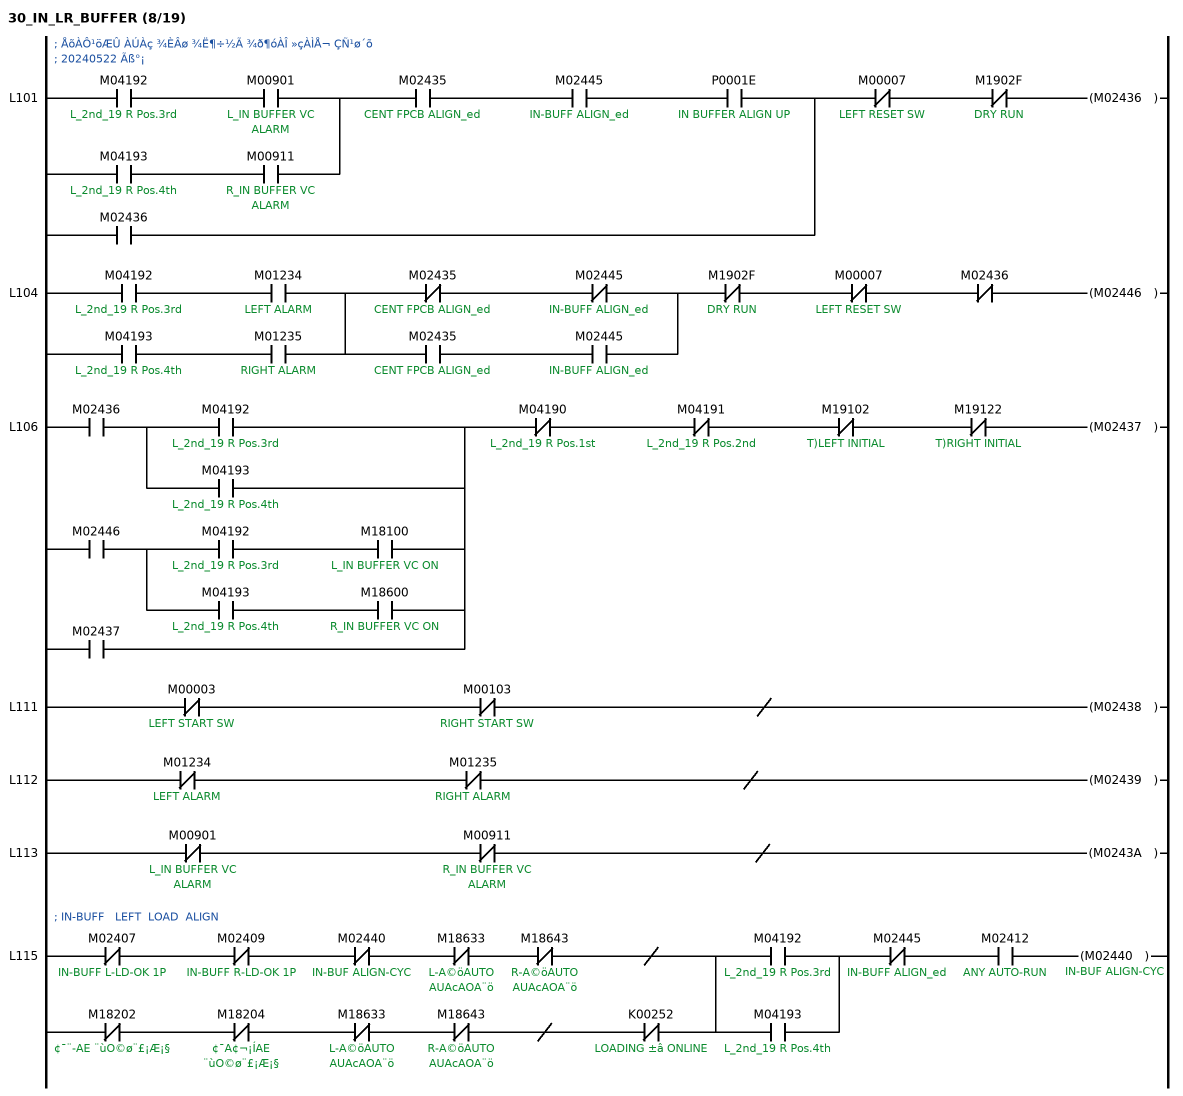
[picture p216: 30_IN_LR_BUFFER rungs L101-L115]
// ÅõÀÔ¹öÆÛ ÀÚÀç ¾ÈÂø ¾Ë¶÷½Ã ¾ð¶óÀÎ »çÀÌÅ¬ ÇÑ¹ø´õ
; L101
LOAD      M04192	// L_2nd_19 R Pos.3rd
AND       M00901	// L_IN BUFFER VC ALARM
LOAD      M04193	// L_2nd_19 R Pos.4th 
AND       M00911	// R_IN BUFFER VC ALARM
OR LOAD
AND       M02435	// CENT FPCB ALIGN_ed
AND       M02445	// IN-BUFF ALIGN_ed
AND       P0001E	// IN BUFFER ALIGN UP
OR        M02436
AND NOT   M00007	// LEFT RESET SW
AND NOT   M1902F	// DRY RUN
OUT       M02436
// output comment: 20240522 Ãß°¡
; L104
LOAD      M04192	// L_2nd_19 R Pos.3rd
AND       M01234	// LEFT ALARM
LOAD      M04193	// L_2nd_19 R Pos.4th 
AND       M01235	// RIGHT ALARM
OR LOAD
LOAD NOT  M02435	// CENT FPCB ALIGN_ed
AND NOT   M02445	// IN-BUFF ALIGN_ed
LOAD      M02435	// CENT FPCB ALIGN_ed
AND       M02445	// IN-BUFF ALIGN_ed
OR LOAD
AND LOAD
AND NOT   M1902F	// DRY RUN
AND NOT   M00007	// LEFT RESET SW
AND NOT   M02436
OUT       M02446
; L106
LOAD      M02436
LOAD      M04192	// L_2nd_19 R Pos.3rd
OR        M04193	// L_2nd_19 R Pos.4th 
AND LOAD
LOAD      M02446
LOAD      M04192	// L_2nd_19 R Pos.3rd
AND       M18100	// L_IN BUFFER VC ON
LOAD      M04193	// L_2nd_19 R Pos.4th 
AND       M18600	// R_IN BUFFER VC ON
OR LOAD
AND LOAD
OR LOAD
OR        M02437
AND NOT   M04190	// L_2nd_19 R Pos.1st 
AND NOT   M04191	// L_2nd_19 R Pos.2nd
AND NOT   M19102	// T)LEFT INITIAL
AND NOT   M19122	// T)RIGHT INITIAL
OUT       M02437
; L111
LOAD NOT  M00003	// LEFT START SW
AND NOT   M00103	// RIGHT START SW
NOT
OUT       M02438
; L112
LOAD NOT  M01234	// LEFT ALARM
AND NOT   M01235	// RIGHT ALARM
NOT
OUT       M02439
; L113
LOAD NOT  M00901	// L_IN BUFFER VC ALARM
AND NOT   M00911	// R_IN BUFFER VC ALARM
NOT
OUT       M0243A
// IN-BUFF   LEFT  LOAD  ALIGN
; L115
LOAD NOT  M02407	// IN-BUFF L-LD-OK 1P
AND NOT   M02409	// IN-BUFF R-LD-OK 1P
AND NOT   M02440	// IN-BUF ALIGN-CYC
AND NOT   M18633	// L-A©öAUTO AUAcAOA¨ö
AND NOT   M18643	// R-A©öAUTO AUAcAOA¨ö
NOT
LOAD NOT  M18202	// ¢¯¨­AE ¨ùO©ø¨£¡Æ¡§
AND NOT   M18204	// ¢¯A¢¬¡ÍAE ¨ùO©ø¨£¡Æ¡§
AND NOT   M18633	// L-A©öAUTO AUAcAOA¨ö
AND NOT   M18643	// R-A©öAUTO AUAcAOA¨ö
NOT
AND NOT   K00252	// LOADING ±â ONLINE
OR LOAD
LOAD      M04192	// L_2nd_19 R Pos.3rd
OR        M04193	// L_2nd_19 R Pos.4th 
AND LOAD
AND NOT   M02445	// IN-BUFF ALIGN_ed
AND       M02412	// ANY AUTO-RUN
OUT       M02440	// IN-BUF ALIGN-CYC

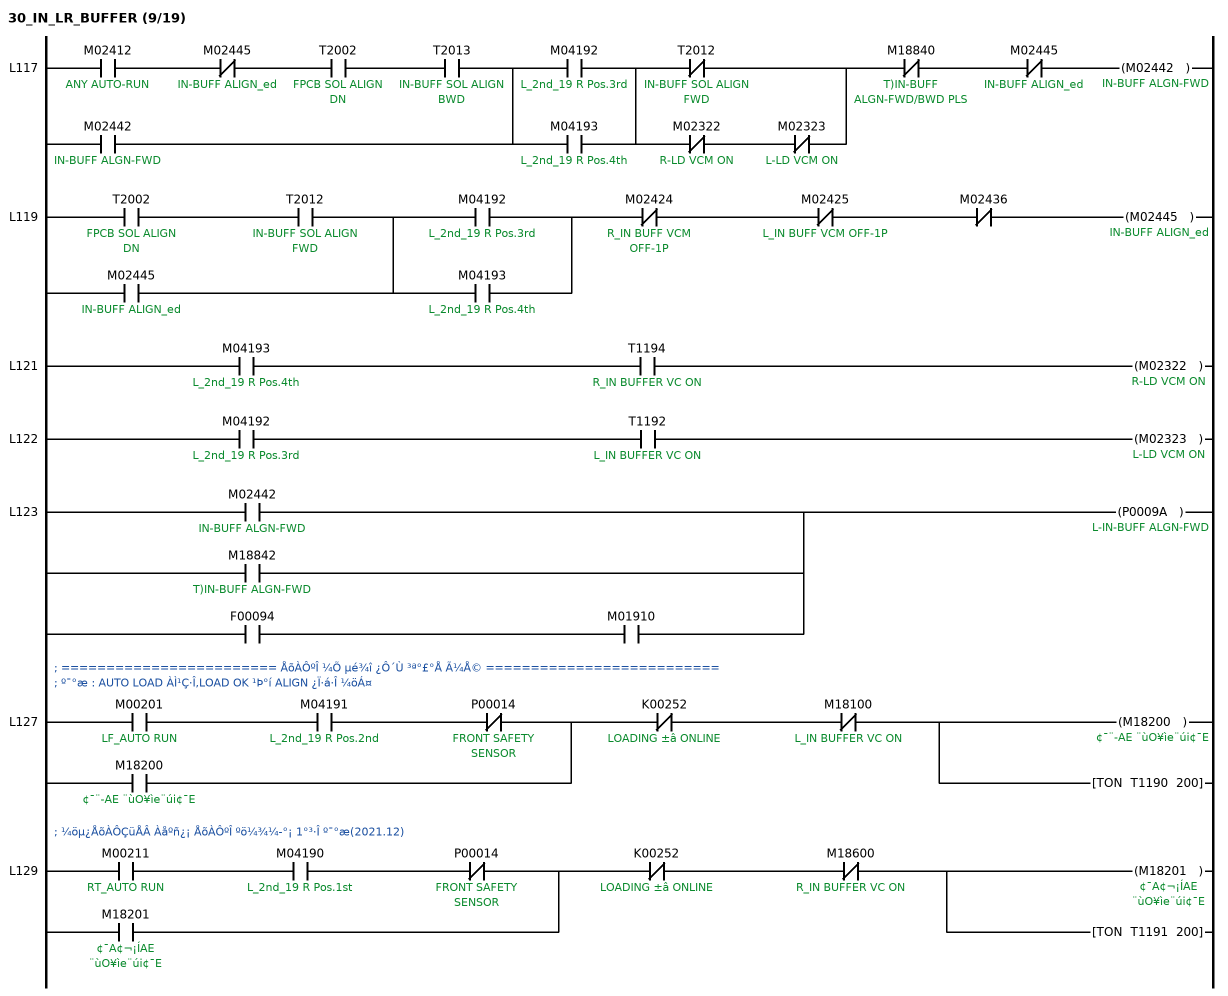
; L117
LOAD      M02412	// ANY AUTO-RUN
AND NOT   M02445	// IN-BUFF ALIGN_ed
AND       T2002	// FPCB SOL ALIGN        DN
AND       T2013	// IN-BUFF SOL ALIGN BWD
OR        M02442	// IN-BUFF ALGN-FWD
LOAD      M04192	// L_2nd_19 R Pos.3rd
OR        M04193	// L_2nd_19 R Pos.4th 
AND LOAD
LOAD NOT  T2012	// IN-BUFF SOL ALIGN FWD
LOAD NOT  M02322	// R-LD VCM ON
AND NOT   M02323	// L-LD VCM ON
OR LOAD
AND LOAD
AND NOT   M18840	// T)IN-BUFF ALGN-FWD/BWD PLS
AND NOT   M02445	// IN-BUFF ALIGN_ed
OUT       M02442	// IN-BUFF ALGN-FWD
; L119
LOAD      T2002	// FPCB SOL ALIGN        DN
AND       T2012	// IN-BUFF SOL ALIGN FWD
OR        M02445	// IN-BUFF ALIGN_ed
LOAD      M04192	// L_2nd_19 R Pos.3rd
OR        M04193	// L_2nd_19 R Pos.4th 
AND LOAD
AND NOT   M02424	// R_IN BUFF VCM OFF-1P
AND NOT   M02425	// L_IN BUFF VCM OFF-1P
AND NOT   M02436
OUT       M02445	// IN-BUFF ALIGN_ed
; L121
LOAD      M04193	// L_2nd_19 R Pos.4th 
AND       T1194	// R_IN BUFFER VC ON
OUT       M02322	// R-LD VCM ON
; L122
LOAD      M04192	// L_2nd_19 R Pos.3rd
AND       T1192	// L_IN BUFFER VC ON
OUT       M02323	// L-LD VCM ON
; L123
LOAD      M02442	// IN-BUFF ALGN-FWD
OR        M18842	// T)IN-BUFF ALGN-FWD
LOAD      F00094
AND       M01910
OR LOAD
OUT       P0009A	// L-IN-BUFF ALGN-FWD
// ======================== ÅõÀÔºÎ ¼Õ µé¾î ¿Ô´Ù ³ª°£°Å Ã¼Å© ==========================
// 
// º¯°æ : AUTO LOAD ÀÌ¹Ç·Î,LOAD OK ¹Þ°í ALIGN ¿Ï·á·Î ¼öÁ¤
; L127
LOAD      M00201	// LF_AUTO RUN
AND       M04191	// L_2nd_19 R Pos.2nd
AND NOT   P00014	// FRONT SAFETY SENSOR
OR        M18200	// ¢¯¨­AE ¨ùO¥ìe¨úi¢¯E
AND NOT   K00252	// LOADING ±â ONLINE
AND NOT   M18100	// L_IN BUFFER VC ON
OUT       M18200	// ¢¯¨­AE ¨ùO¥ìe¨úi¢¯E
TON       T1190 200
; L129
LOAD      M00211	// RT_AUTO RUN
AND       M04190	// L_2nd_19 R Pos.1st 
AND NOT   P00014	// FRONT SAFETY SENSOR
OR        M18201	// ¢¯A¢¬¡ÍAE ¨ùO¥ìe¨úi¢¯E
AND NOT   K00252	// LOADING ±â ONLINE
AND NOT   M18600	// R_IN BUFFER VC ON
OUT       M18201	// ¢¯A¢¬¡ÍAE ¨ùO¥ìe¨úi¢¯E
TON       T1191 200
// output comment: ¼öµ¿ÅõÀÔÇüÅÂ Àåºñ¿¡ ÅõÀÔºÎ ºö¼¾¼­°¡ 1°³·Î º¯°æ(2021.12)

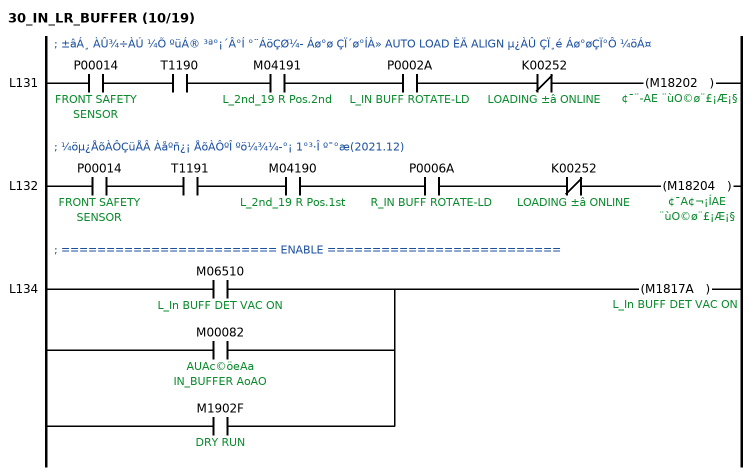
; L131
LOAD      P00014	// FRONT SAFETY SENSOR
AND       T1190
AND       M04191	// L_2nd_19 R Pos.2nd
AND       P0002A	// L_IN BUFF ROTATE-LD
AND NOT   K00252	// LOADING ±â ONLINE
OUT       M18202	// ¢¯¨­AE ¨ùO©ø¨£¡Æ¡§
// output comment: ±âÁ¸ ÀÛ¾÷ÀÚ ¼Õ ºüÁ® ³ª°¡´Â°Í °¨ÁöÇØ¼­ Áø°ø ÇÏ´ø°ÍÀ» AUTO LOAD ÈÄ ALIGN µ¿ÀÛ ÇÏ¸é Áø°øÇÏ°Ô ¼öÁ¤
; L132
LOAD      P00014	// FRONT SAFETY SENSOR
AND       T1191
AND       M04190	// L_2nd_19 R Pos.1st 
AND       P0006A	// R_IN BUFF ROTATE-LD
AND NOT   K00252	// LOADING ±â ONLINE
OUT       M18204	// ¢¯A¢¬¡ÍAE ¨ùO©ø¨£¡Æ¡§
// output comment: ¼öµ¿ÅõÀÔÇüÅÂ Àåºñ¿¡ ÅõÀÔºÎ ºö¼¾¼­°¡ 1°³·Î º¯°æ(2021.12)
// ======================== ENABLE ==========================
; L134
LOAD      M06510	// L_In BUFF DET VAC ON
OR        M00082	// AUAc©öeAa IN_BUFFER AoAO 
OR        M1902F	// DRY RUN
OUT       M1817A	// L_In BUFF DET VAC ON

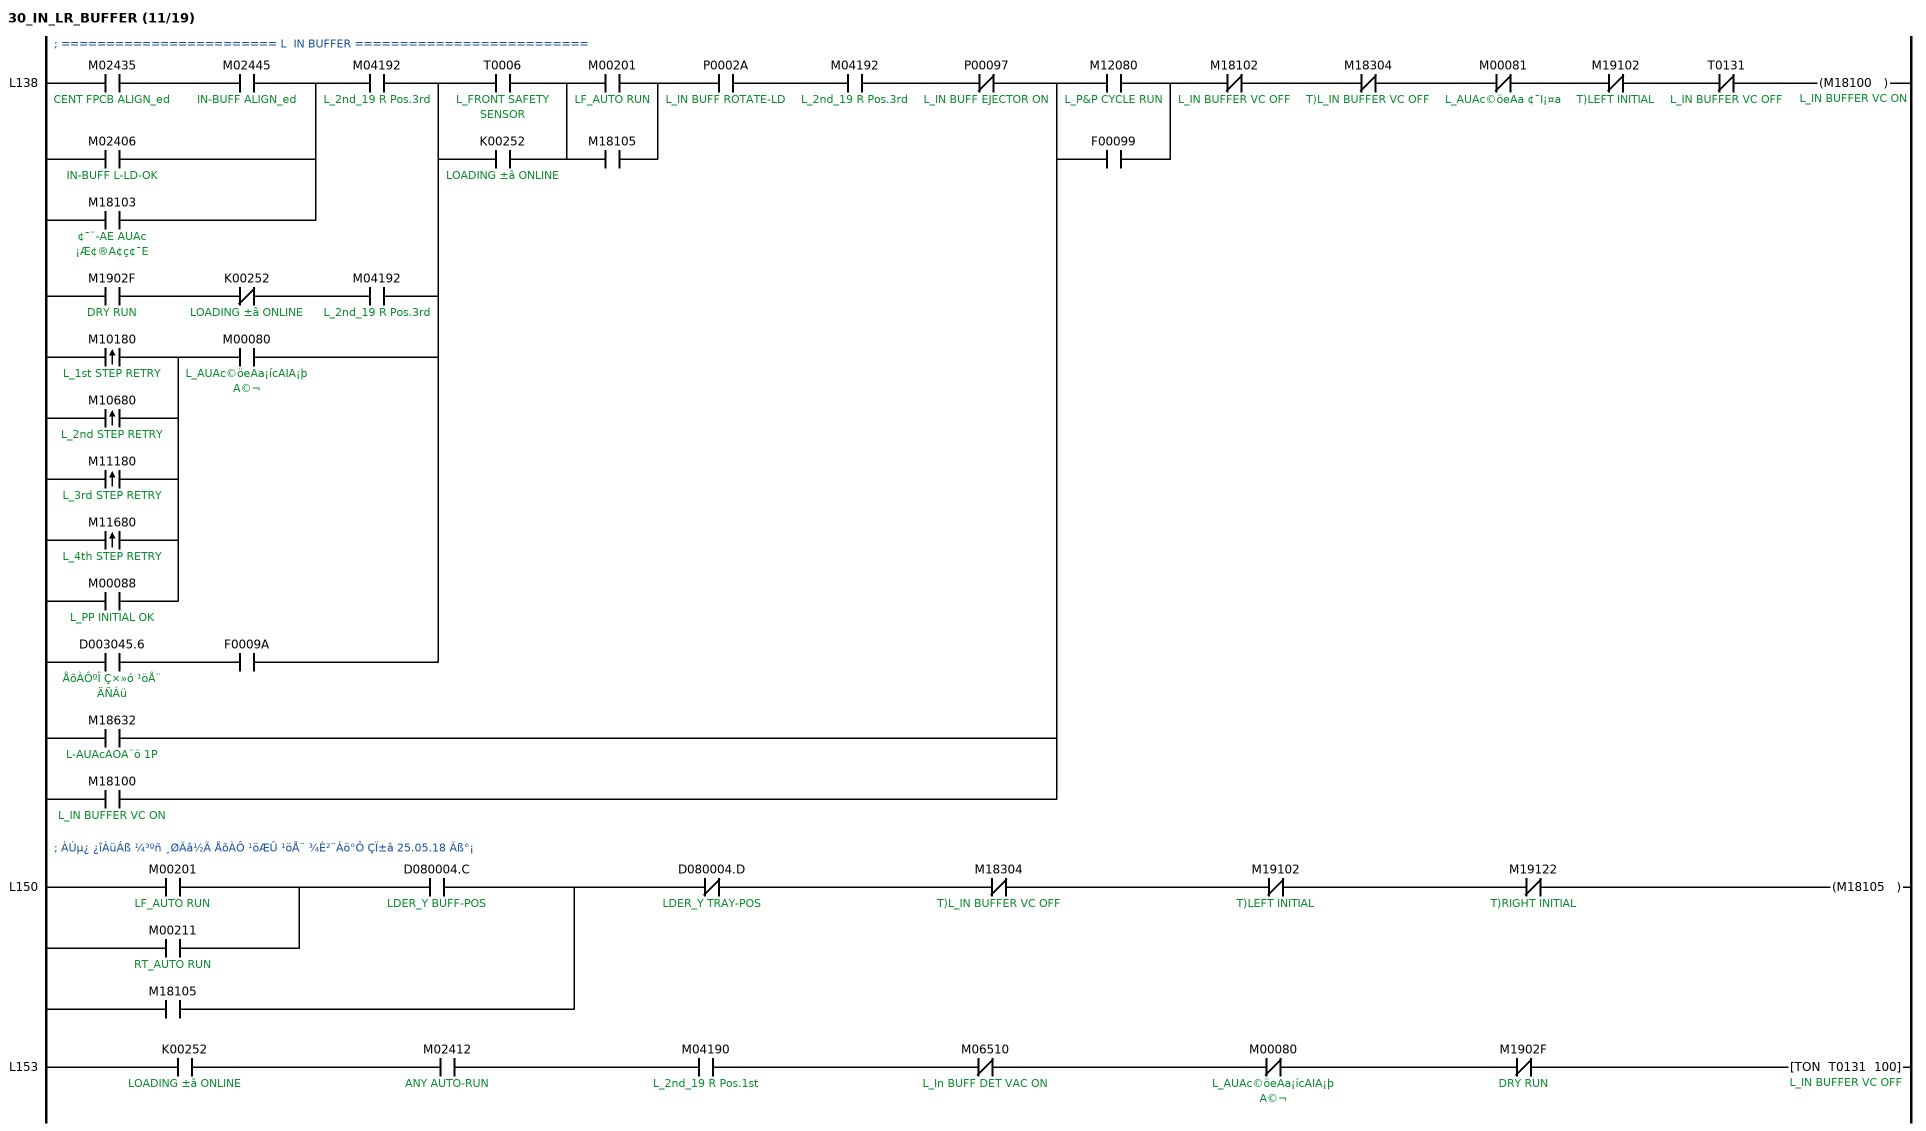
// ======================== L  IN BUFFER ==========================
; L138
LOAD      M02435	// CENT FPCB ALIGN_ed
AND       M02445	// IN-BUFF ALIGN_ed
OR        M02406	// IN-BUFF L-LD-OK
OR        M18103	// ¢¯¨­AE AUAc ¡Æ¢®A¢ç¢¯E
AND       M04192	// L_2nd_19 R Pos.3rd
LOAD      M1902F	// DRY RUN
AND NOT   K00252	// LOADING ±â ONLINE
AND       M04192	// L_2nd_19 R Pos.3rd
OR LOAD
LOADP     M10180	// L_1st STEP RETRY
ORP       M10680	// L_2nd STEP RETRY
ORP       M11180	// L_3rd STEP RETRY
ORP       M11680	// L_4th STEP RETRY
OR        M00088	// L_PP INITIAL OK
AND       M00080	// L_AUAc©öeAa¡ícAIA¡þA©¬
OR LOAD
LOAD      D003045.6	// ÅõÀÔºÎ Ç×»ó ¹öÅ¨ ÄÑÁü
AND       F0009A
OR LOAD
LOAD      T0006	// L_FRONT SAFETY SENSOR
OR        K00252	// LOADING ±â ONLINE
AND LOAD
LOAD      M00201	// LF_AUTO RUN
OR        M18105
AND LOAD
AND       P0002A	// L_IN BUFF ROTATE-LD
AND       M04192	// L_2nd_19 R Pos.3rd
AND NOT   P00097	// L_IN BUFF EJECTOR ON
OR        M18632	// L-AUAcAOA¨ö 1P
OR        M18100	// L_IN BUFFER VC ON
LOAD      M12080	// L_P&P CYCLE RUN
OR        F00099
AND LOAD
AND NOT   M18102	// L_IN BUFFER VC OFF
AND NOT   M18304	// T)L_IN BUFFER VC OFF
AND NOT   M00081	// L_AUAc©öeAa ¢¯I¡¤a
AND NOT   M19102	// T)LEFT INITIAL
AND NOT   T0131	// L_IN BUFFER VC OFF
OUT       M18100	// L_IN BUFFER VC ON
; L150
LOAD      M00201	// LF_AUTO RUN
OR        M00211	// RT_AUTO RUN
AND       D080004.C	// LDER_Y BUFF-POS
OR        M18105
AND NOT   D080004.D	// LDER_Y TRAY-POS
AND NOT   M18304	// T)L_IN BUFFER VC OFF
AND NOT   M19102	// T)LEFT INITIAL
AND NOT   M19122	// T)RIGHT INITIAL
OUT       M18105
// output comment: ÀÚµ¿ ¿îÀüÁß ¼³ºñ ¸ØÃâ½Ã ÅõÀÔ ¹öÆÛ ¹öÅ¨ ¾È²¨Áö°Ô ÇÏ±â 25.05.18 Ãß°¡
; L153
LOAD      K00252	// LOADING ±â ONLINE
AND       M02412	// ANY AUTO-RUN
AND       M04190	// L_2nd_19 R Pos.1st 
AND NOT   M06510	// L_In BUFF DET VAC ON
AND NOT   M00080	// L_AUAc©öeAa¡ícAIA¡þA©¬
AND NOT   M1902F	// DRY RUN
TON       T0131 100	// L_IN BUFFER VC OFF

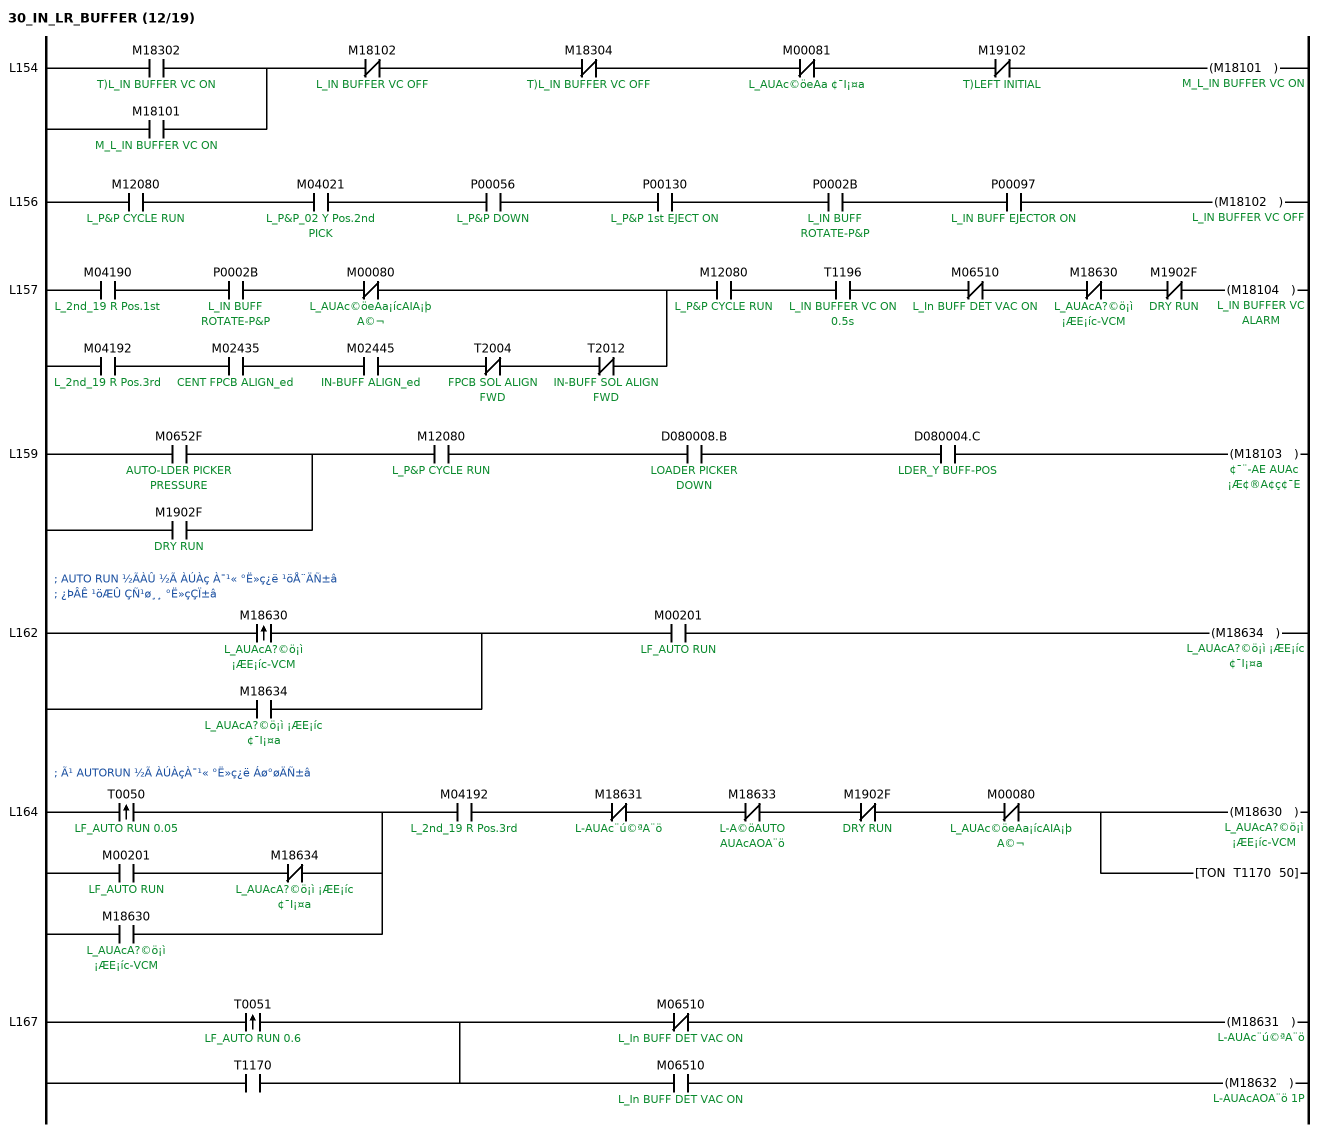
; L154
LOAD      M18302	// T)L_IN BUFFER VC ON
OR        M18101	// M_L_IN BUFFER VC ON
AND NOT   M18102	// L_IN BUFFER VC OFF
AND NOT   M18304	// T)L_IN BUFFER VC OFF
AND NOT   M00081	// L_AUAc©öeAa ¢¯I¡¤a
AND NOT   M19102	// T)LEFT INITIAL
OUT       M18101	// M_L_IN BUFFER VC ON
; L156
LOAD      M12080	// L_P&P CYCLE RUN
AND       M04021	// L_P&P_02 Y Pos.2nd PICK
AND       P00056	// L_P&P DOWN
AND       P00130	// L_P&P 1st EJECT ON
AND       P0002B	// L_IN BUFF ROTATE-P&P
AND       P00097	// L_IN BUFF EJECTOR ON
OUT       M18102	// L_IN BUFFER VC OFF
; L157
LOAD      M04190	// L_2nd_19 R Pos.1st 
AND       P0002B	// L_IN BUFF ROTATE-P&P
AND NOT   M00080	// L_AUAc©öeAa¡ícAIA¡þA©¬
LOAD      M04192	// L_2nd_19 R Pos.3rd
AND       M02435	// CENT FPCB ALIGN_ed
AND       M02445	// IN-BUFF ALIGN_ed
AND NOT   T2004	// FPCB SOL ALIGN         FWD
AND NOT   T2012	// IN-BUFF SOL ALIGN FWD
OR LOAD
AND       M12080	// L_P&P CYCLE RUN
AND       T1196	// L_IN BUFFER VC ON 0.5s
AND NOT   M06510	// L_In BUFF DET VAC ON
AND NOT   M18630	// L_AUAcA?©ö¡ì ¡ÆE¡íc-VCM
AND NOT   M1902F	// DRY RUN
OUT       M18104	// L_IN BUFFER VC ALARM
; L159
LOAD      M0652F	// AUTO-LDER PICKER PRESSURE
OR        M1902F	// DRY RUN
AND       M12080	// L_P&P CYCLE RUN
AND       D080008.B	// LOADER PICKER DOWN
AND       D080004.C	// LDER_Y BUFF-POS
OUT       M18103	// ¢¯¨­AE AUAc ¡Æ¢®A¢ç¢¯E
// AUTO RUN ½ÃÀÛ ½Ã ÀÚÀç À¯¹« °Ë»ç¿ë ¹öÅ¨ÄÑ±â
; L162
LOADP     M18630	// L_AUAcA?©ö¡ì ¡ÆE¡íc-VCM
OR        M18634	// L_AUAcA?©ö¡ì ¡ÆE¡íc ¢¯I¡¤a
AND       M00201	// LF_AUTO RUN
OUT       M18634	// L_AUAcA?©ö¡ì ¡ÆE¡íc ¢¯I¡¤a
// output comment: ¿ÞÂÊ ¹öÆÛ ÇÑ¹ø¸¸ °Ë»çÇÏ±â
; L164
LOADP     T0050	// LF_AUTO RUN 0.05
LOAD      M00201	// LF_AUTO RUN
AND NOT   M18634	// L_AUAcA?©ö¡ì ¡ÆE¡íc ¢¯I¡¤a
OR LOAD
OR        M18630	// L_AUAcA?©ö¡ì ¡ÆE¡íc-VCM
AND       M04192	// L_2nd_19 R Pos.3rd
AND NOT   M18631	// L-AUAc¨ú©ªA¨ö
AND NOT   M18633	// L-A©öAUTO AUAcAOA¨ö
AND NOT   M1902F	// DRY RUN
AND NOT   M00080	// L_AUAc©öeAa¡ícAIA¡þA©¬
OUT       M18630	// L_AUAcA?©ö¡ì ¡ÆE¡íc-VCM
TON       T1170 50
// output comment: Ã¹ AUTORUN ½Ã ÀÚÀçÀ¯¹« °Ë»ç¿ë Áø°øÄÑ±â
; L167
LOADP     T0051	// LF_AUTO RUN 0.6
OR        T1170
MPUSH
AND NOT   M06510	// L_In BUFF DET VAC ON
OUT       M18631	// L-AUAc¨ú©ªA¨ö
MPOP
AND       M06510	// L_In BUFF DET VAC ON
OUT       M18632	// L-AUAcAOA¨ö 1P

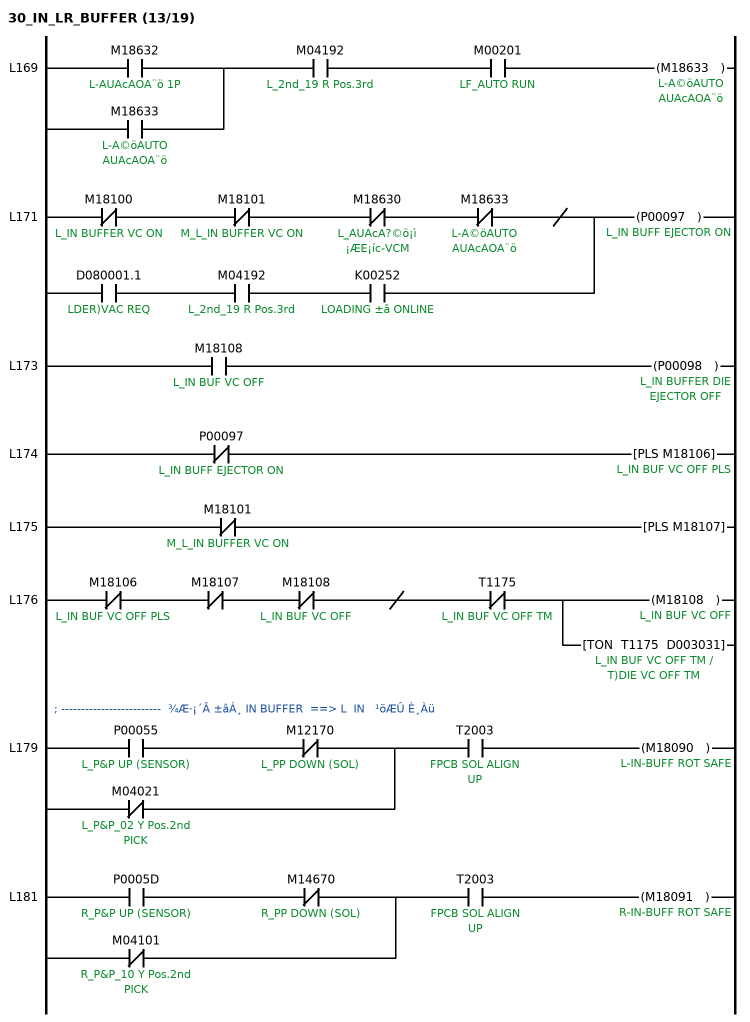
; L169
LOAD      M18632	// L-AUAcAOA¨ö 1P
OR        M18633	// L-A©öAUTO AUAcAOA¨ö
AND       M04192	// L_2nd_19 R Pos.3rd
AND       M00201	// LF_AUTO RUN
OUT       M18633	// L-A©öAUTO AUAcAOA¨ö
; L171
LOAD NOT  M18100	// L_IN BUFFER VC ON
AND NOT   M18101	// M_L_IN BUFFER VC ON
AND NOT   M18630	// L_AUAcA?©ö¡ì ¡ÆE¡íc-VCM
AND NOT   M18633	// L-A©öAUTO AUAcAOA¨ö
NOT
LOAD      D080001.1	// LDER)VAC REQ
AND       M04192	// L_2nd_19 R Pos.3rd
AND       K00252	// LOADING ±â ONLINE
OR LOAD
OUT       P00097	// L_IN BUFF EJECTOR ON
; L173
LOAD      M18108	// L_IN BUF VC OFF
OUT       P00098	// L_IN BUFFER DIE EJECTOR OFF
; L174
LOAD NOT  P00097	// L_IN BUFF EJECTOR ON
OUTP      M18106	// L_IN BUF VC OFF PLS
; L175
LOAD NOT  M18101	// M_L_IN BUFFER VC ON
OUTP      M18107
; L176
LOAD NOT  M18106	// L_IN BUF VC OFF PLS
AND NOT   M18107
AND NOT   M18108	// L_IN BUF VC OFF
NOT
AND NOT   T1175	// L_IN BUF VC OFF TM
OUT       M18108	// L_IN BUF VC OFF
TON       T1175 D003031	// L_IN BUF VC OFF TM / T)DIE VC OFF TM
// -------------------------  ¾Æ·¡´Â ±âÁ¸ IN BUFFER  ==> L  IN   ¹öÆÛ È¸Àü
; L179
LOAD      P00055	// L_P&P UP (SENSOR)
AND NOT   M12170	// L_PP DOWN (SOL)
OR NOT    M04021	// L_P&P_02 Y Pos.2nd PICK
AND       T2003	// FPCB SOL ALIGN         UP
OUT       M18090	// L-IN-BUFF ROT SAFE
; L181
LOAD      P0005D	// R_P&P UP (SENSOR)
AND NOT   M14670	// R_PP DOWN (SOL)
OR NOT    M04101	// R_P&P_10 Y Pos.2nd PICK
AND       T2003	// FPCB SOL ALIGN         UP
OUT       M18091	// R-IN-BUFF ROT SAFE

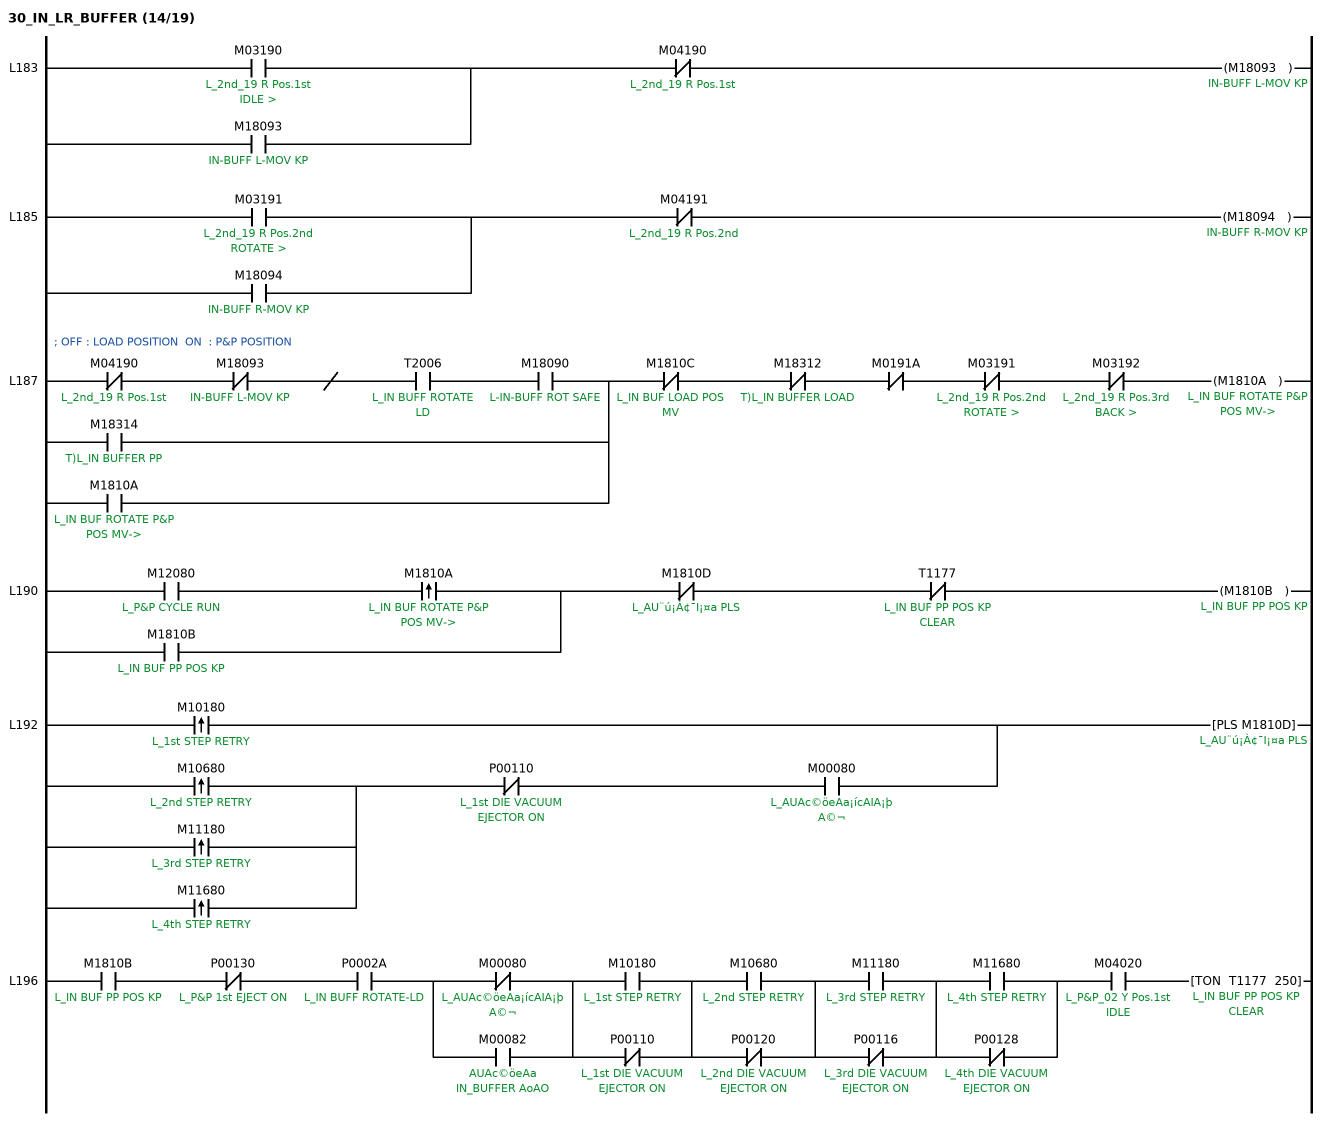
; L183
LOAD      M03190	// L_2nd_19 R Pos.1st IDLE >
OR        M18093	// IN-BUFF L-MOV KP
AND NOT   M04190	// L_2nd_19 R Pos.1st 
OUT       M18093	// IN-BUFF L-MOV KP
; L185
LOAD      M03191	// L_2nd_19 R Pos.2nd ROTATE >
OR        M18094	// IN-BUFF R-MOV KP
AND NOT   M04191	// L_2nd_19 R Pos.2nd
OUT       M18094	// IN-BUFF R-MOV KP
; L187
LOAD NOT  M04190	// L_2nd_19 R Pos.1st 
AND NOT   M18093	// IN-BUFF L-MOV KP
NOT
AND       T2006	// L_IN BUFF ROTATE     LD
AND       M18090	// L-IN-BUFF ROT SAFE
OR        M18314	// T)L_IN BUFFER PP
OR        M1810A	// L_IN BUF ROTATE P&P POS MV->
AND NOT   M1810C	// L_IN BUF LOAD POS MV
AND NOT   M18312	// T)L_IN BUFFER LOAD
AND NOT   M0191A
AND NOT   M03191	// L_2nd_19 R Pos.2nd ROTATE >
AND NOT   M03192	// L_2nd_19 R Pos.3rd BACK >
OUT       M1810A	// L_IN BUF ROTATE P&P POS MV->
// output comment: OFF : LOAD POSITION  ON  : P&P POSITION
; L190
LOAD      M12080	// L_P&P CYCLE RUN
ANDP      M1810A	// L_IN BUF ROTATE P&P POS MV->
OR        M1810B	// L_IN BUF PP POS KP
AND NOT   M1810D	// L_AU¨ú¡À¢¯I¡¤a PLS
AND NOT   T1177	// L_IN BUF PP POS KP CLEAR
OUT       M1810B	// L_IN BUF PP POS KP
; L192
LOADP     M10180	// L_1st STEP RETRY
LOADP     M10680	// L_2nd STEP RETRY
ORP       M11180	// L_3rd STEP RETRY
ORP       M11680	// L_4th STEP RETRY
AND NOT   P00110	// L_1st DIE VACUUM EJECTOR ON
AND       M00080	// L_AUAc©öeAa¡ícAIA¡þA©¬
OR LOAD
OUTP      M1810D	// L_AU¨ú¡À¢¯I¡¤a PLS
; L196
LOAD      M1810B	// L_IN BUF PP POS KP
AND NOT   P00130	// L_P&P 1st EJECT ON
AND       P0002A	// L_IN BUFF ROTATE-LD
LOAD NOT  M00080	// L_AUAc©öeAa¡ícAIA¡þA©¬
OR        M00082	// AUAc©öeAa IN_BUFFER AoAO 
AND LOAD
LOAD      M10180	// L_1st STEP RETRY
OR NOT    P00110	// L_1st DIE VACUUM EJECTOR ON
AND LOAD
LOAD      M10680	// L_2nd STEP RETRY
OR NOT    P00120	// L_2nd DIE VACUUM EJECTOR ON
AND LOAD
LOAD      M11180	// L_3rd STEP RETRY
OR NOT    P00116	// L_3rd DIE VACUUM EJECTOR ON
AND LOAD
LOAD      M11680	// L_4th STEP RETRY
OR NOT    P00128	// L_4th DIE VACUUM EJECTOR ON
AND LOAD
AND       M04020	// L_P&P_02 Y Pos.1st IDLE
TON       T1177 250	// L_IN BUF PP POS KP CLEAR

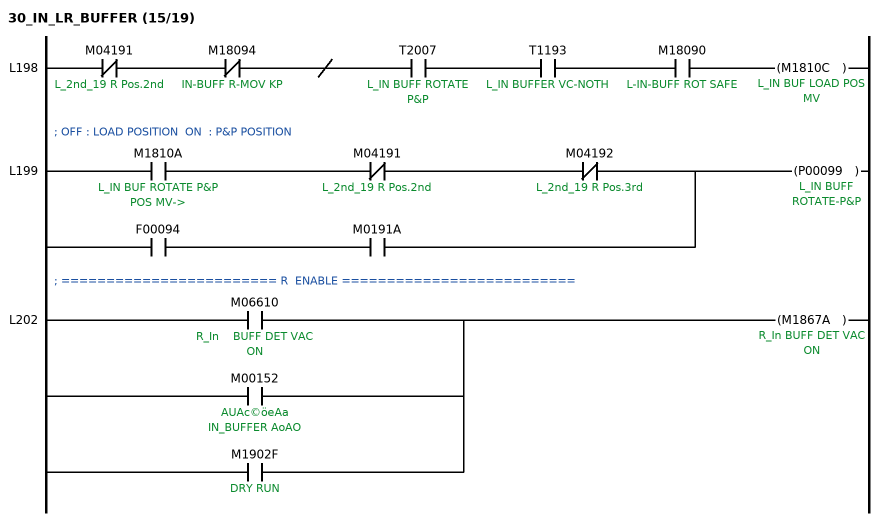
; L198
LOAD NOT  M04191	// L_2nd_19 R Pos.2nd
AND NOT   M18094	// IN-BUFF R-MOV KP
NOT
AND       T2007	// L_IN BUFF ROTATE      P&P
AND       T1193	// L_IN BUFFER VC-NOTH
AND       M18090	// L-IN-BUFF ROT SAFE
OUT       M1810C	// L_IN BUF LOAD POS MV
; L199
LOAD      M1810A	// L_IN BUF ROTATE P&P POS MV->
AND NOT   M04191	// L_2nd_19 R Pos.2nd
AND NOT   M04192	// L_2nd_19 R Pos.3rd
LOAD      F00094
AND       M0191A
OR LOAD
OUT       P00099	// L_IN BUFF ROTATE-P&P
// output comment: OFF : LOAD POSITION  ON  : P&P POSITION
// ======================== R  ENABLE ==========================
; L202
LOAD      M06610	// R_In    BUFF DET VAC ON
OR        M00152	// AUAc©öeAa IN_BUFFER AoAO 
OR        M1902F	// DRY RUN
OUT       M1867A	// R_In BUFF DET VAC ON

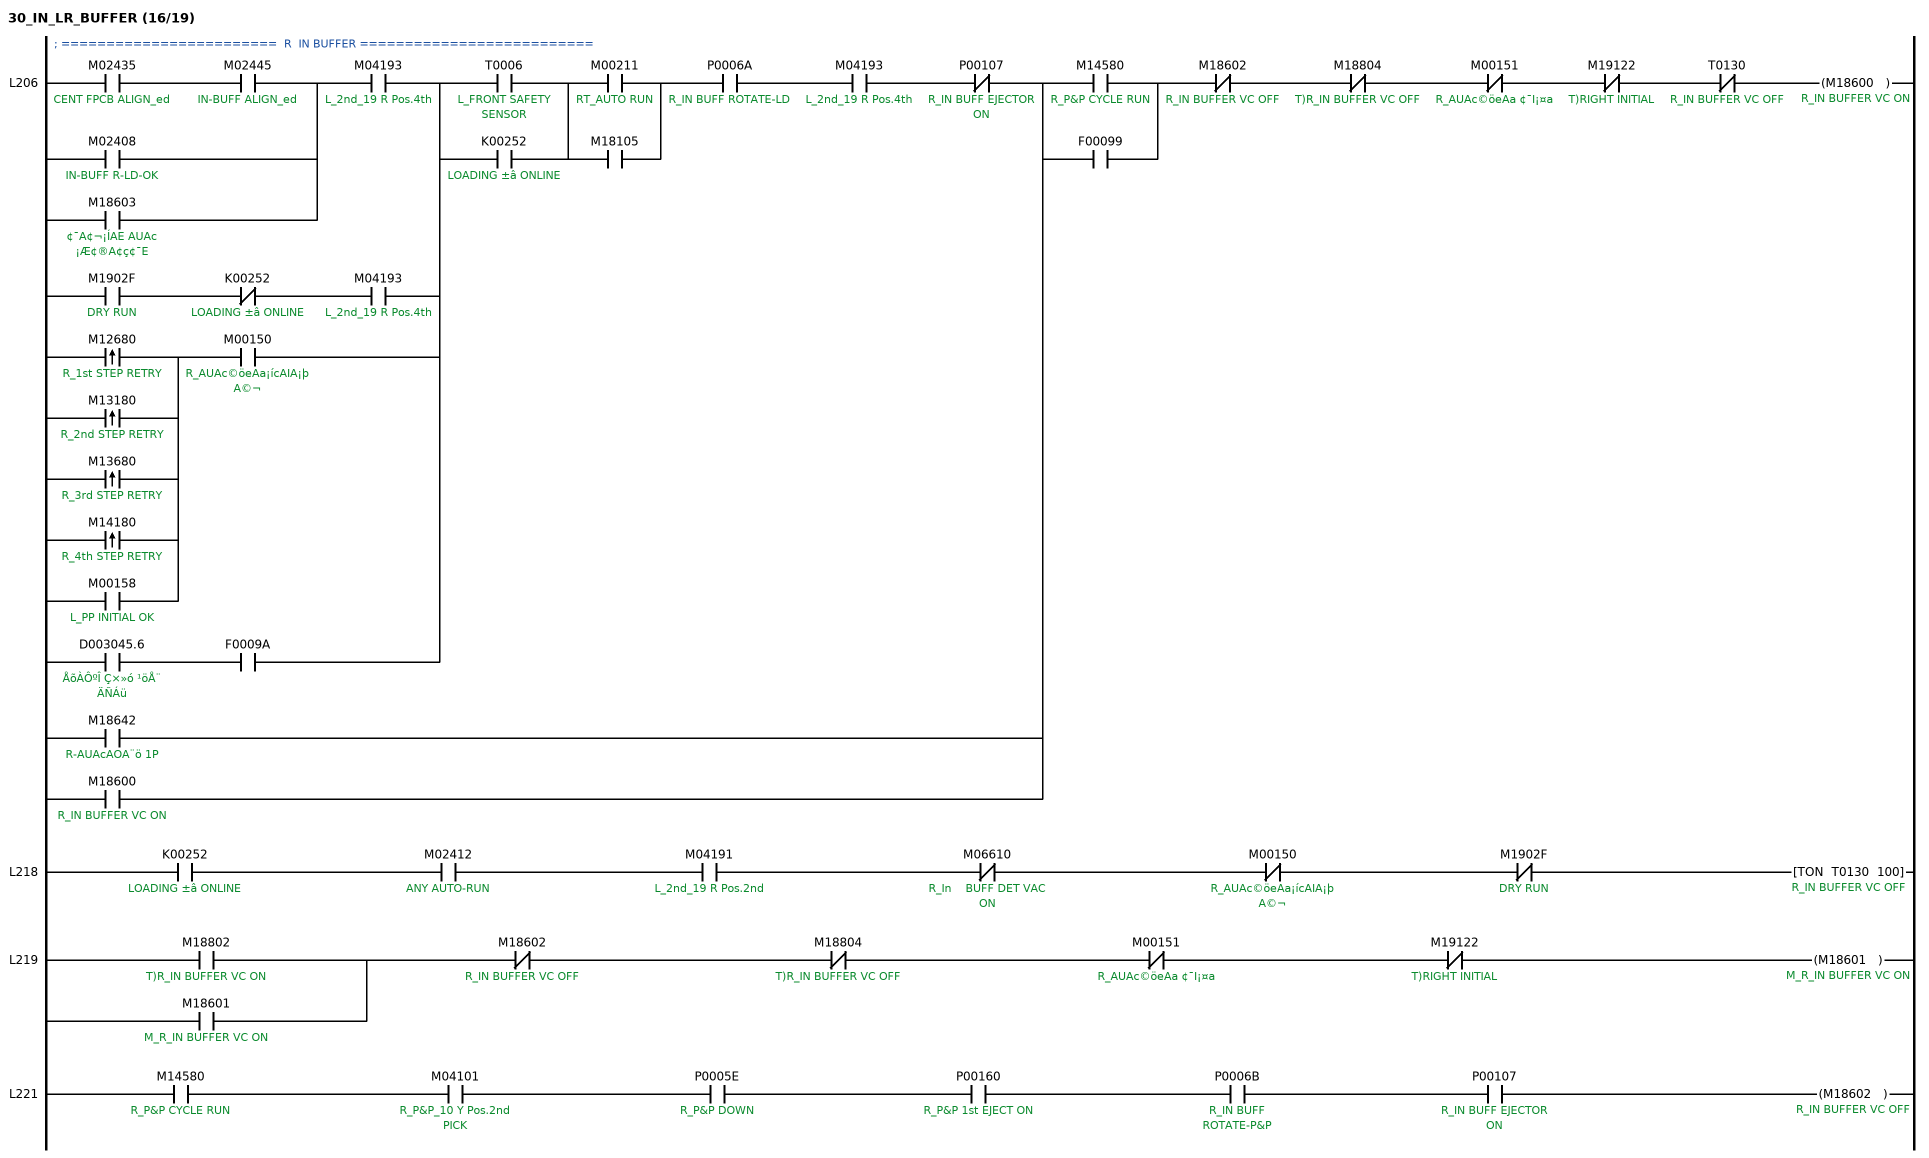
// ========================  R  IN BUFFER ==========================
; L206
LOAD      M02435	// CENT FPCB ALIGN_ed
AND       M02445	// IN-BUFF ALIGN_ed
OR        M02408	// IN-BUFF R-LD-OK
OR        M18603	// ¢¯A¢¬¡ÍAE AUAc ¡Æ¢®A¢ç¢¯E
AND       M04193	// L_2nd_19 R Pos.4th 
LOAD      M1902F	// DRY RUN
AND NOT   K00252	// LOADING ±â ONLINE
AND       M04193	// L_2nd_19 R Pos.4th 
OR LOAD
LOADP     M12680	// R_1st STEP RETRY
ORP       M13180	// R_2nd STEP RETRY
ORP       M13680	// R_3rd STEP RETRY
ORP       M14180	// R_4th STEP RETRY
OR        M00158	// L_PP INITIAL OK
AND       M00150	// R_AUAc©öeAa¡ícAIA¡þA©¬
OR LOAD
LOAD      D003045.6	// ÅõÀÔºÎ Ç×»ó ¹öÅ¨ ÄÑÁü
AND       F0009A
OR LOAD
LOAD      T0006	// L_FRONT SAFETY SENSOR
OR        K00252	// LOADING ±â ONLINE
AND LOAD
LOAD      M00211	// RT_AUTO RUN
OR        M18105
AND LOAD
AND       P0006A	// R_IN BUFF ROTATE-LD
AND       M04193	// L_2nd_19 R Pos.4th 
AND NOT   P00107	// R_IN BUFF EJECTOR ON
OR        M18642	// R-AUAcAOA¨ö 1P
OR        M18600	// R_IN BUFFER VC ON
LOAD      M14580	// R_P&P CYCLE RUN
OR        F00099
AND LOAD
AND NOT   M18602	// R_IN BUFFER VC OFF
AND NOT   M18804	// T)R_IN BUFFER VC OFF
AND NOT   M00151	// R_AUAc©öeAa ¢¯I¡¤a
AND NOT   M19122	// T)RIGHT INITIAL
AND NOT   T0130	// R_IN BUFFER VC OFF
OUT       M18600	// R_IN BUFFER VC ON
; L218
LOAD      K00252	// LOADING ±â ONLINE
AND       M02412	// ANY AUTO-RUN
AND       M04191	// L_2nd_19 R Pos.2nd
AND NOT   M06610	// R_In    BUFF DET VAC ON
AND NOT   M00150	// R_AUAc©öeAa¡ícAIA¡þA©¬
AND NOT   M1902F	// DRY RUN
TON       T0130 100	// R_IN BUFFER VC OFF
; L219
LOAD      M18802	// T)R_IN BUFFER VC ON
OR        M18601	// M_R_IN BUFFER VC ON
AND NOT   M18602	// R_IN BUFFER VC OFF
AND NOT   M18804	// T)R_IN BUFFER VC OFF
AND NOT   M00151	// R_AUAc©öeAa ¢¯I¡¤a
AND NOT   M19122	// T)RIGHT INITIAL
OUT       M18601	// M_R_IN BUFFER VC ON
; L221
LOAD      M14580	// R_P&P CYCLE RUN
AND       M04101	// R_P&P_10 Y Pos.2nd PICK
AND       P0005E	// R_P&P DOWN
AND       P00160	// R_P&P 1st EJECT ON
AND       P0006B	// R_IN BUFF ROTATE-P&P
AND       P00107	// R_IN BUFF EJECTOR ON
OUT       M18602	// R_IN BUFFER VC OFF

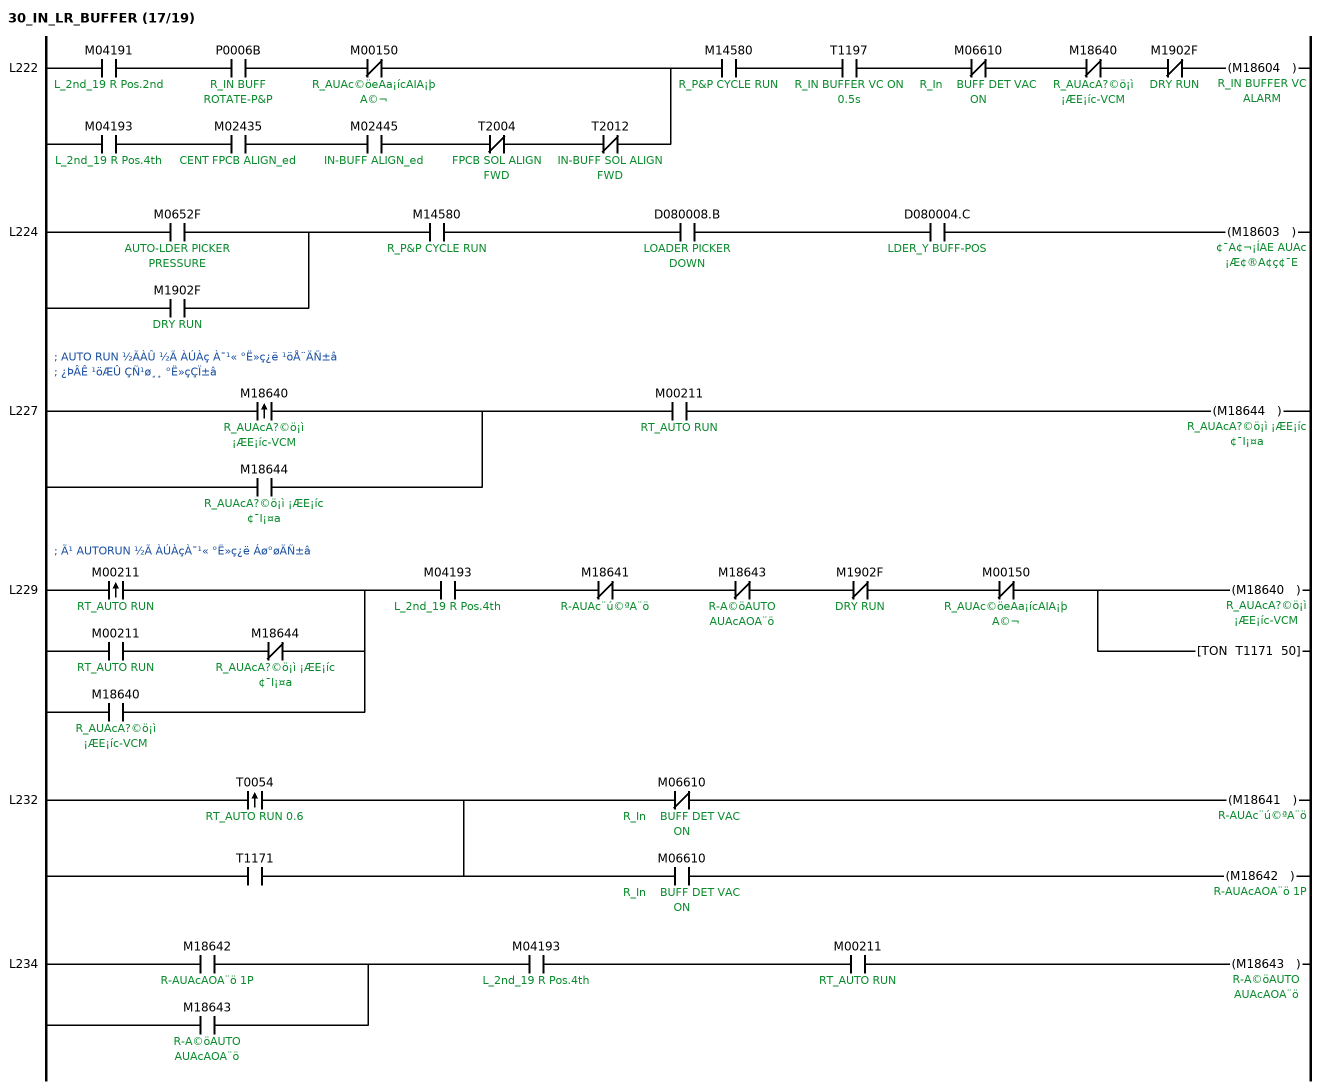
; L222
LOAD      M04191	// L_2nd_19 R Pos.2nd
AND       P0006B	// R_IN BUFF ROTATE-P&P
AND NOT   M00150	// R_AUAc©öeAa¡ícAIA¡þA©¬
LOAD      M04193	// L_2nd_19 R Pos.4th 
AND       M02435	// CENT FPCB ALIGN_ed
AND       M02445	// IN-BUFF ALIGN_ed
AND NOT   T2004	// FPCB SOL ALIGN         FWD
AND NOT   T2012	// IN-BUFF SOL ALIGN FWD
OR LOAD
AND       M14580	// R_P&P CYCLE RUN
AND       T1197	// R_IN BUFFER VC ON 0.5s
AND NOT   M06610	// R_In    BUFF DET VAC ON
AND NOT   M18640	// R_AUAcA?©ö¡ì ¡ÆE¡íc-VCM
AND NOT   M1902F	// DRY RUN
OUT       M18604	// R_IN BUFFER VC ALARM
; L224
LOAD      M0652F	// AUTO-LDER PICKER PRESSURE
OR        M1902F	// DRY RUN
AND       M14580	// R_P&P CYCLE RUN
AND       D080008.B	// LOADER PICKER DOWN
AND       D080004.C	// LDER_Y BUFF-POS
OUT       M18603	// ¢¯A¢¬¡ÍAE AUAc ¡Æ¢®A¢ç¢¯E
// AUTO RUN ½ÃÀÛ ½Ã ÀÚÀç À¯¹« °Ë»ç¿ë ¹öÅ¨ÄÑ±â
; L227
LOADP     M18640	// R_AUAcA?©ö¡ì ¡ÆE¡íc-VCM
OR        M18644	// R_AUAcA?©ö¡ì ¡ÆE¡íc ¢¯I¡¤a
AND       M00211	// RT_AUTO RUN
OUT       M18644	// R_AUAcA?©ö¡ì ¡ÆE¡íc ¢¯I¡¤a
// output comment: ¿ÞÂÊ ¹öÆÛ ÇÑ¹ø¸¸ °Ë»çÇÏ±â
; L229
LOADP     M00211	// RT_AUTO RUN
LOAD      M00211	// RT_AUTO RUN
AND NOT   M18644	// R_AUAcA?©ö¡ì ¡ÆE¡íc ¢¯I¡¤a
OR LOAD
OR        M18640	// R_AUAcA?©ö¡ì ¡ÆE¡íc-VCM
AND       M04193	// L_2nd_19 R Pos.4th 
AND NOT   M18641	// R-AUAc¨ú©ªA¨ö
AND NOT   M18643	// R-A©öAUTO AUAcAOA¨ö
AND NOT   M1902F	// DRY RUN
AND NOT   M00150	// R_AUAc©öeAa¡ícAIA¡þA©¬
OUT       M18640	// R_AUAcA?©ö¡ì ¡ÆE¡íc-VCM
TON       T1171 50
// output comment: Ã¹ AUTORUN ½Ã ÀÚÀçÀ¯¹« °Ë»ç¿ë Áø°øÄÑ±â
; L232
LOADP     T0054	// RT_AUTO RUN 0.6
OR        T1171
MPUSH
AND NOT   M06610	// R_In    BUFF DET VAC ON
OUT       M18641	// R-AUAc¨ú©ªA¨ö
MPOP
AND       M06610	// R_In    BUFF DET VAC ON
OUT       M18642	// R-AUAcAOA¨ö 1P
; L234
LOAD      M18642	// R-AUAcAOA¨ö 1P
OR        M18643	// R-A©öAUTO AUAcAOA¨ö
AND       M04193	// L_2nd_19 R Pos.4th 
AND       M00211	// RT_AUTO RUN
OUT       M18643	// R-A©öAUTO AUAcAOA¨ö

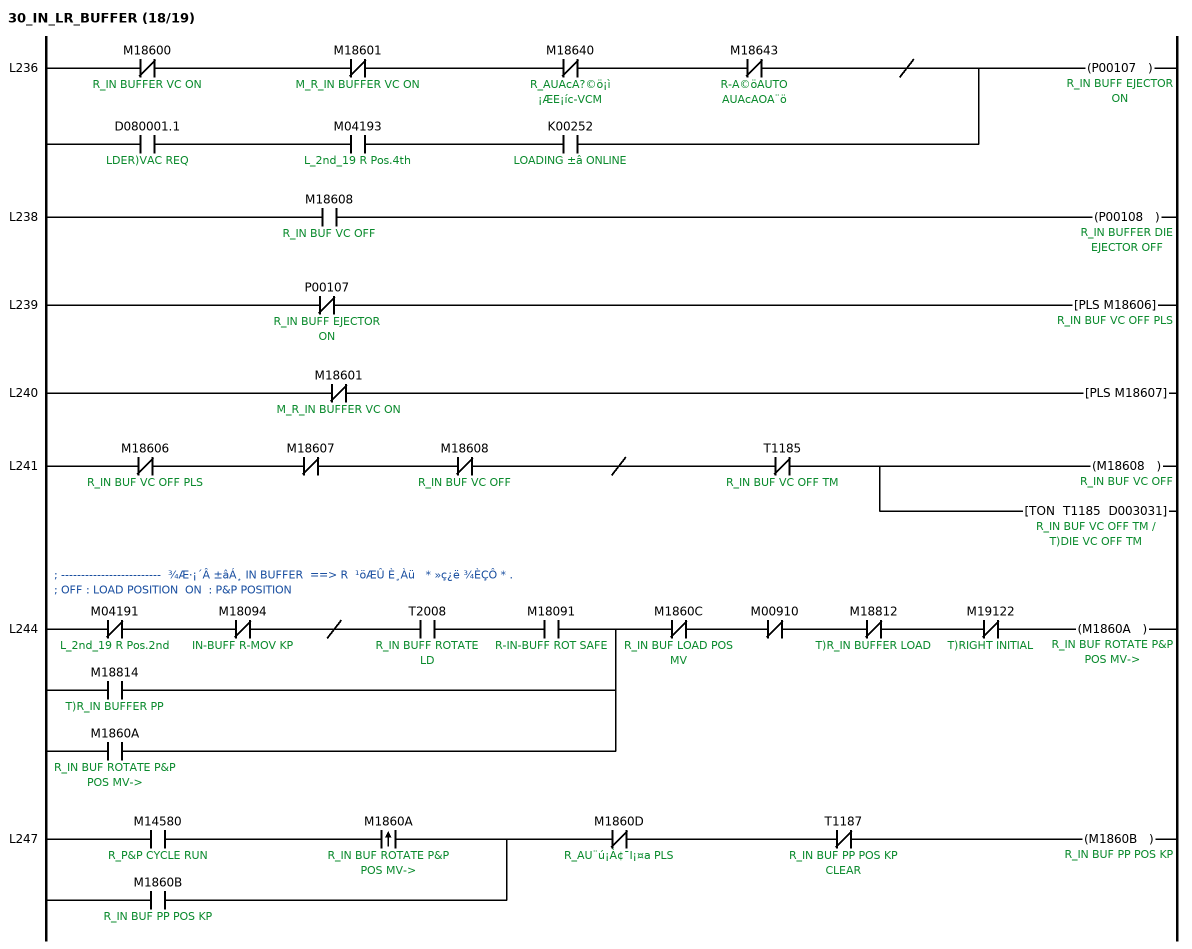
; L236
LOAD NOT  M18600	// R_IN BUFFER VC ON
AND NOT   M18601	// M_R_IN BUFFER VC ON
AND NOT   M18640	// R_AUAcA?©ö¡ì ¡ÆE¡íc-VCM
AND NOT   M18643	// R-A©öAUTO AUAcAOA¨ö
NOT
LOAD      D080001.1	// LDER)VAC REQ
AND       M04193	// L_2nd_19 R Pos.4th 
AND       K00252	// LOADING ±â ONLINE
OR LOAD
OUT       P00107	// R_IN BUFF EJECTOR ON
; L238
LOAD      M18608	// R_IN BUF VC OFF
OUT       P00108	// R_IN BUFFER DIE EJECTOR OFF
; L239
LOAD NOT  P00107	// R_IN BUFF EJECTOR ON
OUTP      M18606	// R_IN BUF VC OFF PLS
; L240
LOAD NOT  M18601	// M_R_IN BUFFER VC ON
OUTP      M18607
; L241
LOAD NOT  M18606	// R_IN BUF VC OFF PLS
AND NOT   M18607
AND NOT   M18608	// R_IN BUF VC OFF
NOT
AND NOT   T1185	// R_IN BUF VC OFF TM
OUT       M18608	// R_IN BUF VC OFF
TON       T1185 D003031	// R_IN BUF VC OFF TM / T)DIE VC OFF TM
// -------------------------  ¾Æ·¡´Â ±âÁ¸ IN BUFFER  ==> R  ¹öÆÛ È¸Àü   * »ç¿ë ¾ÈÇÔ * .
; L244
LOAD NOT  M04191	// L_2nd_19 R Pos.2nd
AND NOT   M18094	// IN-BUFF R-MOV KP
NOT
AND       T2008	// R_IN BUFF ROTATE      LD
AND       M18091	// R-IN-BUFF ROT SAFE
OR        M18814	// T)R_IN BUFFER PP
OR        M1860A	// R_IN BUF ROTATE P&P POS MV->
AND NOT   M1860C	// R_IN BUF LOAD POS MV
AND NOT   M00910
AND NOT   M18812	// T)R_IN BUFFER LOAD
AND NOT   M19122	// T)RIGHT INITIAL
OUT       M1860A	// R_IN BUF ROTATE P&P POS MV->
// output comment: OFF : LOAD POSITION  ON  : P&P POSITION
; L247
LOAD      M14580	// R_P&P CYCLE RUN
ANDP      M1860A	// R_IN BUF ROTATE P&P POS MV->
OR        M1860B	// R_IN BUF PP POS KP
AND NOT   M1860D	// R_AU¨ú¡À¢¯I¡¤a PLS
AND NOT   T1187	// R_IN BUF PP POS KP CLEAR
OUT       M1860B	// R_IN BUF PP POS KP

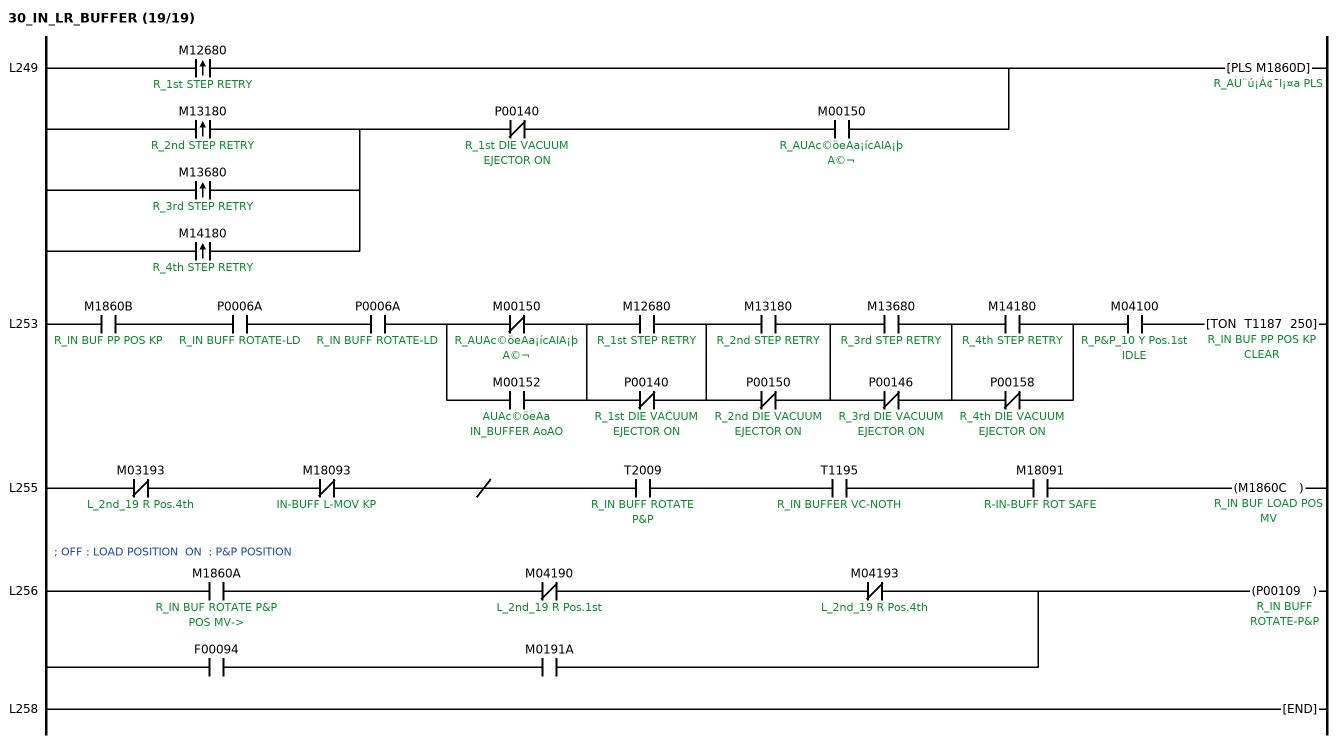
; L249
LOADP     M12680	// R_1st STEP RETRY
LOADP     M13180	// R_2nd STEP RETRY
ORP       M13680	// R_3rd STEP RETRY
ORP       M14180	// R_4th STEP RETRY
AND NOT   P00140	// R_1st DIE VACUUM EJECTOR ON
AND       M00150	// R_AUAc©öeAa¡ícAIA¡þA©¬
OR LOAD
OUTP      M1860D	// R_AU¨ú¡À¢¯I¡¤a PLS
; L253
LOAD      M1860B	// R_IN BUF PP POS KP
AND       P0006A	// R_IN BUFF ROTATE-LD
AND       P0006A	// R_IN BUFF ROTATE-LD
LOAD NOT  M00150	// R_AUAc©öeAa¡ícAIA¡þA©¬
OR        M00152	// AUAc©öeAa IN_BUFFER AoAO 
AND LOAD
LOAD      M12680	// R_1st STEP RETRY
OR NOT    P00140	// R_1st DIE VACUUM EJECTOR ON
AND LOAD
LOAD      M13180	// R_2nd STEP RETRY
OR NOT    P00150	// R_2nd DIE VACUUM EJECTOR ON
AND LOAD
LOAD      M13680	// R_3rd STEP RETRY
OR NOT    P00146	// R_3rd DIE VACUUM EJECTOR ON
AND LOAD
LOAD      M14180	// R_4th STEP RETRY
OR NOT    P00158	// R_4th DIE VACUUM EJECTOR ON
AND LOAD
AND       M04100	// R_P&P_10 Y Pos.1st IDLE
TON       T1187 250	// R_IN BUF PP POS KP CLEAR
; L255
LOAD NOT  M03193	// L_2nd_19 R Pos.4th 
AND NOT   M18093	// IN-BUFF L-MOV KP
NOT
AND       T2009	// R_IN BUFF ROTATE      P&P
AND       T1195	// R_IN BUFFER VC-NOTH
AND       M18091	// R-IN-BUFF ROT SAFE
OUT       M1860C	// R_IN BUF LOAD POS MV
; L256
LOAD      M1860A	// R_IN BUF ROTATE P&P POS MV->
AND NOT   M04190	// L_2nd_19 R Pos.1st 
AND NOT   M04193	// L_2nd_19 R Pos.4th 
LOAD      F00094
AND       M0191A
OR LOAD
OUT       P00109	// R_IN BUFF ROTATE-P&P
// output comment: OFF : LOAD POSITION  ON  : P&P POSITION
; L258
END

PROGRAM 31_OUT_LR_BUFFER (task: ½ºÄµ ÇÁ·Î±×·¥)

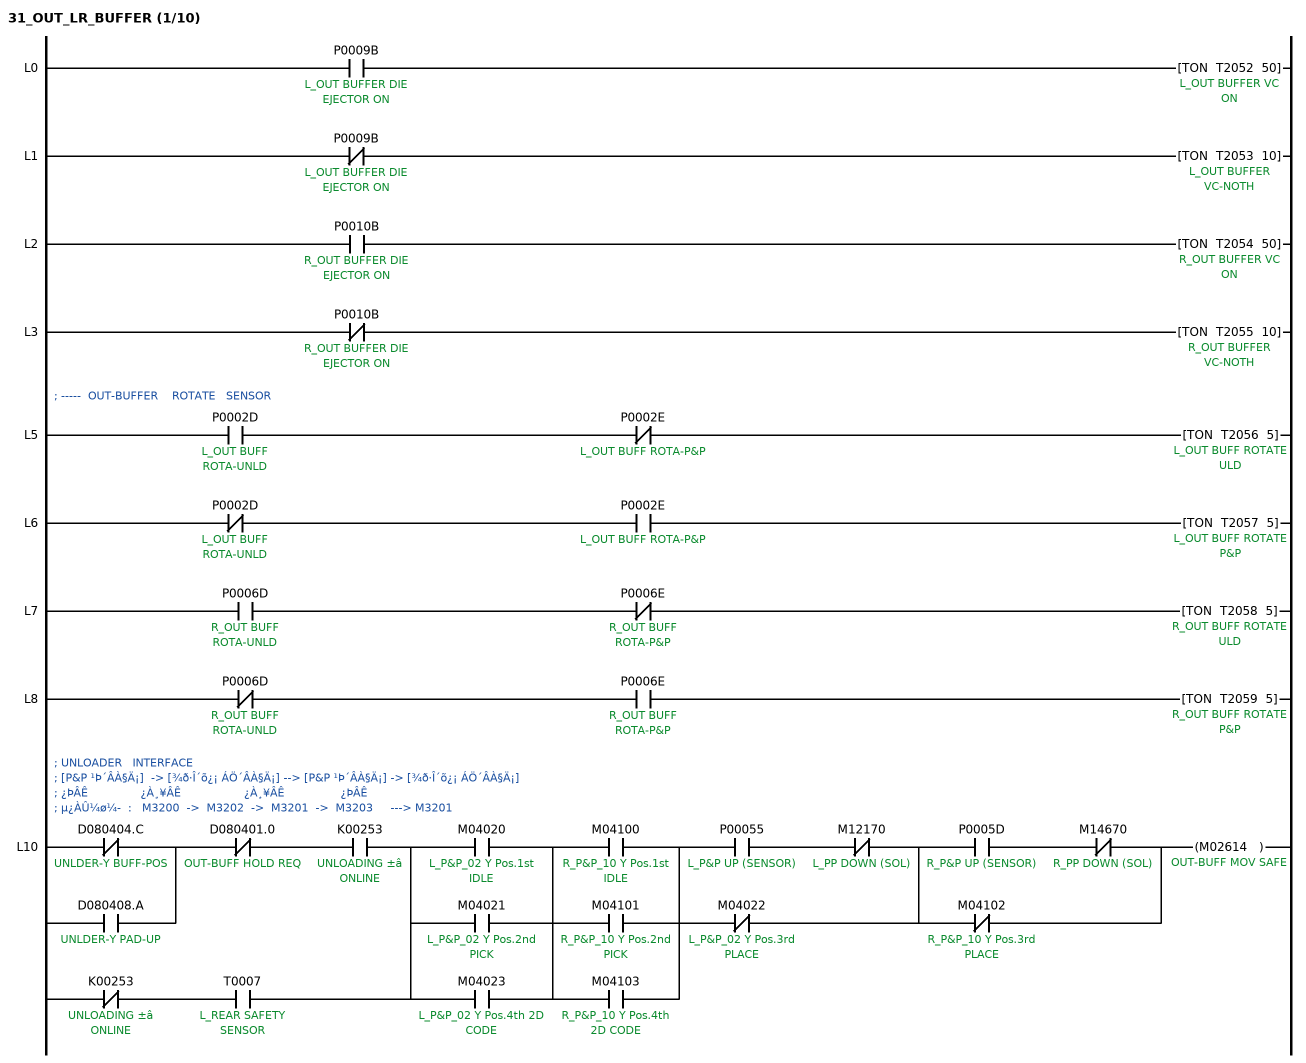
; L0
LOAD      P0009B	// L_OUT BUFFER DIE EJECTOR ON
TON       T2052 50	// L_OUT BUFFER VC ON
; L1
LOAD NOT  P0009B	// L_OUT BUFFER DIE EJECTOR ON
TON       T2053 10	// L_OUT BUFFER VC-NOTH
; L2
LOAD      P0010B	// R_OUT BUFFER DIE EJECTOR ON
TON       T2054 50	// R_OUT BUFFER VC ON
; L3
LOAD NOT  P0010B	// R_OUT BUFFER DIE EJECTOR ON
TON       T2055 10	// R_OUT BUFFER VC-NOTH
// -----  OUT-BUFFER    ROTATE   SENSOR
; L5
LOAD      P0002D	// L_OUT BUFF ROTA-UNLD
AND NOT   P0002E	// L_OUT BUFF ROTA-P&P
TON       T2056 5	// L_OUT BUFF ROTATE     ULD
; L6
LOAD NOT  P0002D	// L_OUT BUFF ROTA-UNLD
AND       P0002E	// L_OUT BUFF ROTA-P&P
TON       T2057 5	// L_OUT BUFF ROTATE      P&P
; L7
LOAD      P0006D	// R_OUT BUFF ROTA-UNLD
AND NOT   P0006E	// R_OUT BUFF ROTA-P&P
TON       T2058 5	// R_OUT BUFF ROTATE      ULD
; L8
LOAD NOT  P0006D	// R_OUT BUFF ROTA-UNLD
AND       P0006E	// R_OUT BUFF ROTA-P&P
TON       T2059 5	// R_OUT BUFF ROTATE      P&P
//  UNLOADER   INTERFACE
//  
//   [P&P ¹Þ´ÂÀ§Ä¡]  -> [¾ð·Î´õ¿¡ ÁÖ´ÂÀ§Ä¡] --> [P&P ¹Þ´ÂÀ§Ä¡] -> [¾ð·Î´õ¿¡ ÁÖ´ÂÀ§Ä¡]
//       ¿ÞÂÊ               ¿À¸¥ÂÊ                  ¿À¸¥ÂÊ                ¿ÞÂÊ
//     
//  µ¿ÀÛ¼ø¼­  :   M3200  ->  M3202  ->  M3201  ->  M3203     ---> M3201
; L10
LOAD NOT  D080404.C	// UNLDER-Y BUFF-POS
OR        D080408.A	// UNLDER-Y PAD-UP
AND NOT   D080401.0	// OUT-BUFF HOLD REQ
AND       K00253	// UNLOADING ±â ONLINE
LOAD NOT  K00253	// UNLOADING ±â ONLINE
AND       T0007	// L_REAR SAFETY SENSOR
OR LOAD
LOAD      M04020	// L_P&P_02 Y Pos.1st IDLE
OR        M04021	// L_P&P_02 Y Pos.2nd PICK
OR        M04023	// L_P&P_02 Y Pos.4th 2D CODE
AND LOAD
LOAD      M04100	// R_P&P_10 Y Pos.1st IDLE
OR        M04101	// R_P&P_10 Y Pos.2nd PICK
OR        M04103	// R_P&P_10 Y Pos.4th 2D CODE
AND LOAD
LOAD      P00055	// L_P&P UP (SENSOR)
AND NOT   M12170	// L_PP DOWN (SOL)
OR NOT    M04022	// L_P&P_02 Y Pos.3rd PLACE
AND LOAD
LOAD      P0005D	// R_P&P UP (SENSOR)
AND NOT   M14670	// R_PP DOWN (SOL)
OR NOT    M04102	// R_P&P_10 Y Pos.3rd PLACE
AND LOAD
OUT       M02614	// OUT-BUFF MOV SAFE

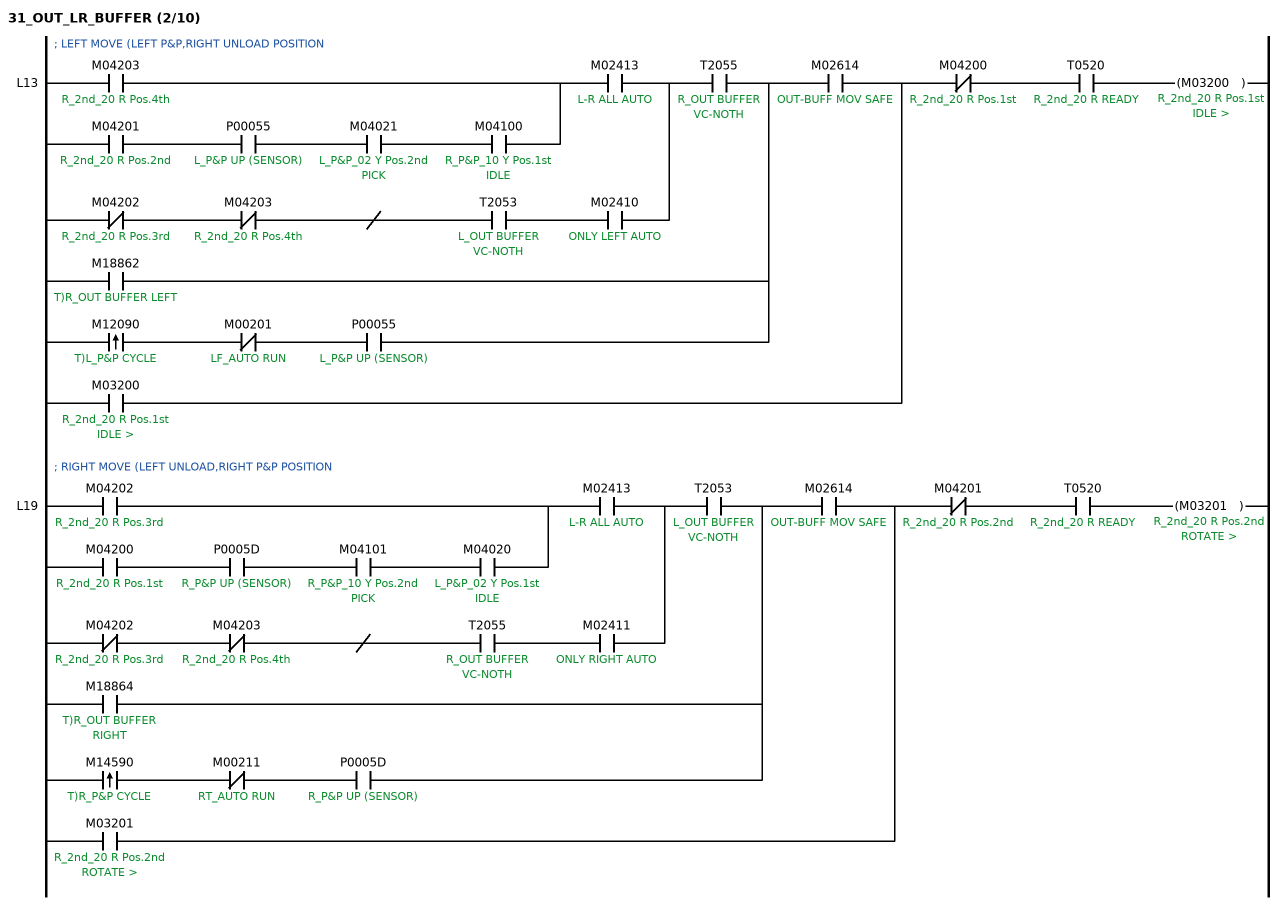
; L13
LOAD      M04203	// R_2nd_20 R Pos.4th 
LOAD      M04201	// R_2nd_20 R Pos.2nd
AND       P00055	// L_P&P UP (SENSOR)
AND       M04021	// L_P&P_02 Y Pos.2nd PICK
AND       M04100	// R_P&P_10 Y Pos.1st IDLE
OR LOAD
AND       M02413	// L-R ALL AUTO
LOAD NOT  M04202	// R_2nd_20 R Pos.3rd
AND NOT   M04203	// R_2nd_20 R Pos.4th 
NOT
AND       T2053	// L_OUT BUFFER VC-NOTH
AND       M02410	// ONLY LEFT AUTO
OR LOAD
AND       T2055	// R_OUT BUFFER VC-NOTH
OR        M18862	// T)R_OUT BUFFER LEFT
LOADP     M12090	// T)L_P&P CYCLE
AND NOT   M00201	// LF_AUTO RUN
AND       P00055	// L_P&P UP (SENSOR)
OR LOAD
AND       M02614	// OUT-BUFF MOV SAFE
OR        M03200	// R_2nd_20 R Pos.1st IDLE >
AND NOT   M04200	// R_2nd_20 R Pos.1st
AND       T0520	// R_2nd_20 R READY
OUT       M03200	// R_2nd_20 R Pos.1st IDLE >
// output comment: LEFT MOVE (LEFT P&P,RIGHT UNLOAD POSITION
; L19
LOAD      M04202	// R_2nd_20 R Pos.3rd
LOAD      M04200	// R_2nd_20 R Pos.1st
AND       P0005D	// R_P&P UP (SENSOR)
AND       M04101	// R_P&P_10 Y Pos.2nd PICK
AND       M04020	// L_P&P_02 Y Pos.1st IDLE
OR LOAD
AND       M02413	// L-R ALL AUTO
LOAD NOT  M04202	// R_2nd_20 R Pos.3rd
AND NOT   M04203	// R_2nd_20 R Pos.4th 
NOT
AND       T2055	// R_OUT BUFFER VC-NOTH
AND       M02411	// ONLY RIGHT AUTO
OR LOAD
AND       T2053	// L_OUT BUFFER VC-NOTH
OR        M18864	// T)R_OUT BUFFER RIGHT
LOADP     M14590	// T)R_P&P CYCLE
AND NOT   M00211	// RT_AUTO RUN
AND       P0005D	// R_P&P UP (SENSOR)
OR LOAD
AND       M02614	// OUT-BUFF MOV SAFE
OR        M03201	// R_2nd_20 R Pos.2nd ROTATE >
AND NOT   M04201	// R_2nd_20 R Pos.2nd
AND       T0520	// R_2nd_20 R READY
OUT       M03201	// R_2nd_20 R Pos.2nd ROTATE >
// output comment: RIGHT MOVE (LEFT UNLOAD,RIGHT P&P POSITION

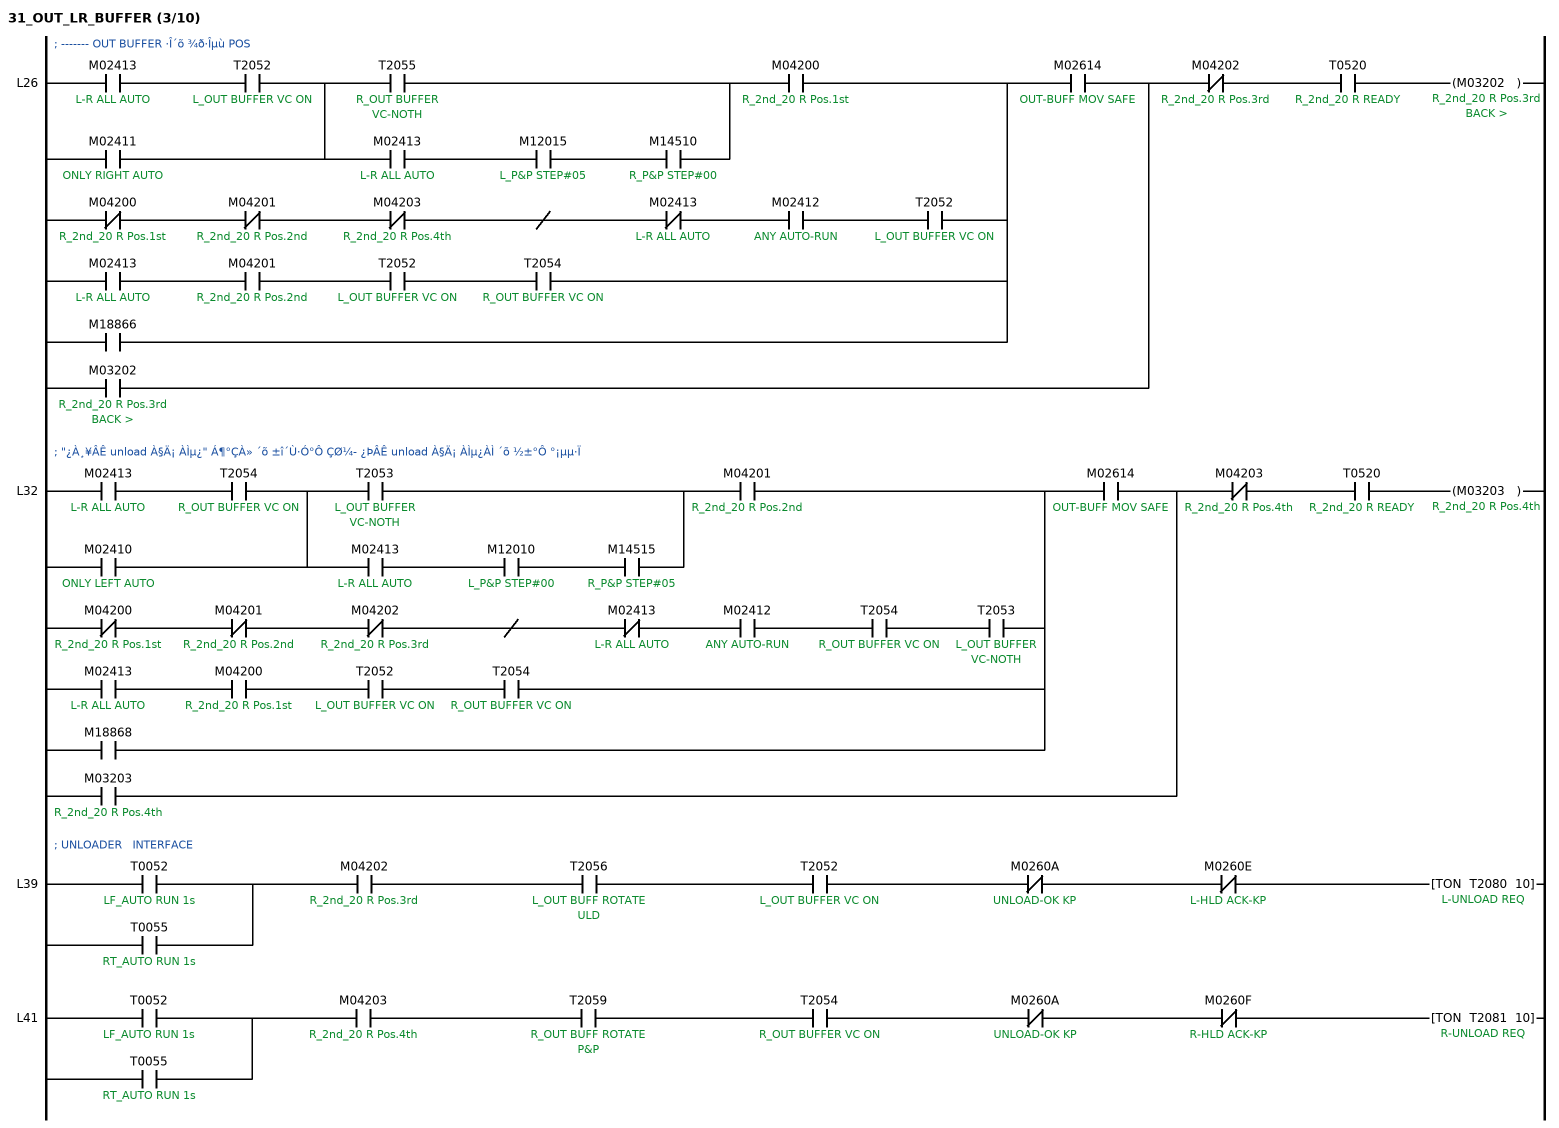
// ------- OUT BUFFER ·Î´õ ¾ð·Îµù POS
; L26
LOAD      M02413	// L-R ALL AUTO
AND       T2052	// L_OUT BUFFER VC ON
OR        M02411	// ONLY RIGHT AUTO
LOAD      T2055	// R_OUT BUFFER VC-NOTH
LOAD      M02413	// L-R ALL AUTO
AND       M12015	// L_P&P STEP#05
AND       M14510	// R_P&P STEP#00
OR LOAD
AND LOAD
AND       M04200	// R_2nd_20 R Pos.1st
LOAD NOT  M04200	// R_2nd_20 R Pos.1st
AND NOT   M04201	// R_2nd_20 R Pos.2nd
AND NOT   M04203	// R_2nd_20 R Pos.4th 
NOT
AND NOT   M02413	// L-R ALL AUTO
AND       M02412	// ANY AUTO-RUN
AND       T2052	// L_OUT BUFFER VC ON
OR LOAD
LOAD      M02413	// L-R ALL AUTO
AND       M04201	// R_2nd_20 R Pos.2nd
AND       T2052	// L_OUT BUFFER VC ON
AND       T2054	// R_OUT BUFFER VC ON
OR LOAD
OR        M18866
AND       M02614	// OUT-BUFF MOV SAFE
OR        M03202	// R_2nd_20 R Pos.3rd BACK >
AND NOT   M04202	// R_2nd_20 R Pos.3rd
AND       T0520	// R_2nd_20 R READY
OUT       M03202	// R_2nd_20 R Pos.3rd BACK >
; L32
LOAD      M02413	// L-R ALL AUTO
AND       T2054	// R_OUT BUFFER VC ON
OR        M02410	// ONLY LEFT AUTO
LOAD      T2053	// L_OUT BUFFER VC-NOTH
LOAD      M02413	// L-R ALL AUTO
AND       M12010	// L_P&P STEP#00
AND       M14515	// R_P&P STEP#05
OR LOAD
AND LOAD
AND       M04201	// R_2nd_20 R Pos.2nd
LOAD NOT  M04200	// R_2nd_20 R Pos.1st
AND NOT   M04201	// R_2nd_20 R Pos.2nd
AND NOT   M04202	// R_2nd_20 R Pos.3rd
NOT
AND NOT   M02413	// L-R ALL AUTO
AND       M02412	// ANY AUTO-RUN
AND       T2054	// R_OUT BUFFER VC ON
AND       T2053	// L_OUT BUFFER VC-NOTH
OR LOAD
LOAD      M02413	// L-R ALL AUTO
AND       M04200	// R_2nd_20 R Pos.1st
AND       T2052	// L_OUT BUFFER VC ON
AND       T2054	// R_OUT BUFFER VC ON
OR LOAD
OR        M18868
AND       M02614	// OUT-BUFF MOV SAFE
OR        M03203	// R_2nd_20 R Pos.4th 
AND NOT   M04203	// R_2nd_20 R Pos.4th 
AND       T0520	// R_2nd_20 R READY
OUT       M03203	// R_2nd_20 R Pos.4th 
// output comment: "¿À¸¥ÂÊ unload À§Ä¡ ÀÌµ¿" Á¶°ÇÀ» ´õ ±î´Ù·Ó°Ô ÇØ¼­ ¿ÞÂÊ unload À§Ä¡ ÀÌµ¿ÀÌ ´õ ½±°Ô °¡µµ·Ï
//  UNLOADER   INTERFACE
; L39
LOAD      T0052	// LF_AUTO RUN 1s
OR        T0055	// RT_AUTO RUN 1s
AND       M04202	// R_2nd_20 R Pos.3rd
AND       T2056	// L_OUT BUFF ROTATE     ULD
AND       T2052	// L_OUT BUFFER VC ON
AND NOT   M0260A	// UNLOAD-OK KP
AND NOT   M0260E	// L-HLD ACK-KP
TON       T2080 10	// L-UNLOAD REQ
; L41
LOAD      T0052	// LF_AUTO RUN 1s
OR        T0055	// RT_AUTO RUN 1s
AND       M04203	// R_2nd_20 R Pos.4th 
AND       T2059	// R_OUT BUFF ROTATE      P&P
AND       T2054	// R_OUT BUFFER VC ON
AND NOT   M0260A	// UNLOAD-OK KP
AND NOT   M0260F	// R-HLD ACK-KP
TON       T2081 10	// R-UNLOAD REQ

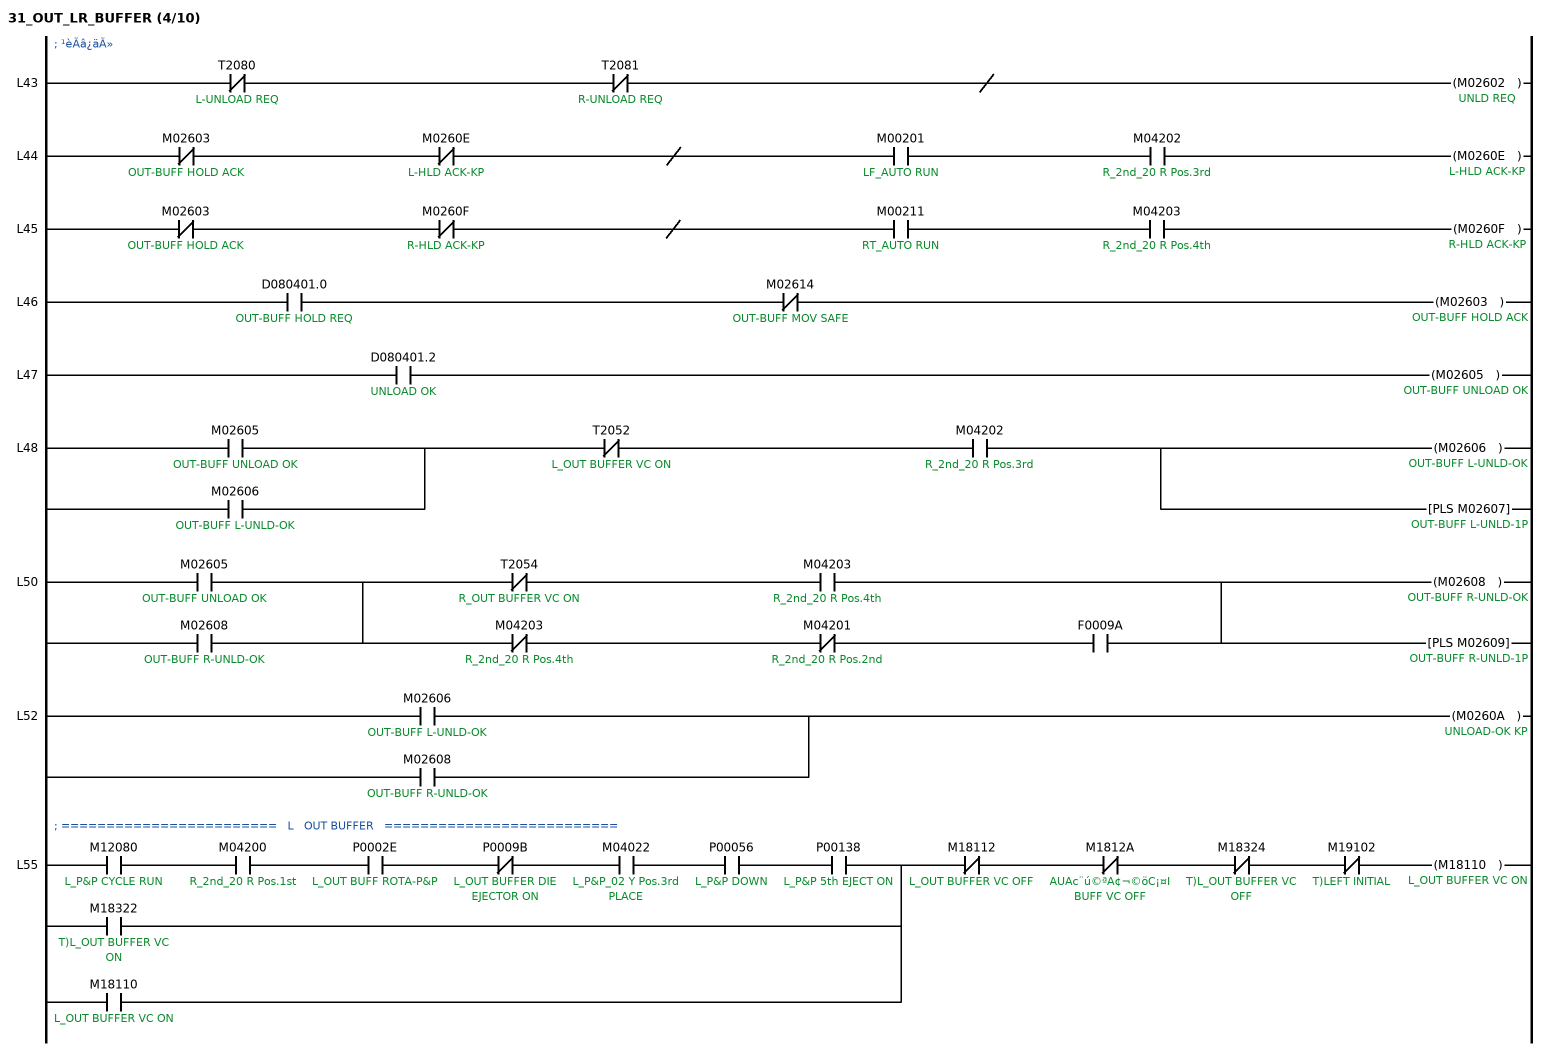
; L43
LOAD NOT  T2080	// L-UNLOAD REQ
AND NOT   T2081	// R-UNLOAD REQ
NOT
OUT       M02602	// UNLD REQ
// output comment: ¹èÃâ¿äÃ»
; L44
LOAD NOT  M02603	// OUT-BUFF HOLD ACK
AND NOT   M0260E	// L-HLD ACK-KP
NOT
AND       M00201	// LF_AUTO RUN
AND       M04202	// R_2nd_20 R Pos.3rd
OUT       M0260E	// L-HLD ACK-KP
; L45
LOAD NOT  M02603	// OUT-BUFF HOLD ACK
AND NOT   M0260F	// R-HLD ACK-KP
NOT
AND       M00211	// RT_AUTO RUN
AND       M04203	// R_2nd_20 R Pos.4th 
OUT       M0260F	// R-HLD ACK-KP
; L46
LOAD      D080401.0	// OUT-BUFF HOLD REQ
AND NOT   M02614	// OUT-BUFF MOV SAFE
OUT       M02603	// OUT-BUFF HOLD ACK
; L47
LOAD      D080401.2	// UNLOAD OK
OUT       M02605	// OUT-BUFF UNLOAD OK
; L48
LOAD      M02605	// OUT-BUFF UNLOAD OK
OR        M02606	// OUT-BUFF L-UNLD-OK
AND NOT   T2052	// L_OUT BUFFER VC ON
AND       M04202	// R_2nd_20 R Pos.3rd
OUT       M02606	// OUT-BUFF L-UNLD-OK
OUTP      M02607	// OUT-BUFF L-UNLD-1P
; L50
LOAD      M02605	// OUT-BUFF UNLOAD OK
OR        M02608	// OUT-BUFF R-UNLD-OK
LOAD NOT  T2054	// R_OUT BUFFER VC ON
AND       M04203	// R_2nd_20 R Pos.4th 
LOAD NOT  M04203	// R_2nd_20 R Pos.4th 
AND NOT   M04201	// R_2nd_20 R Pos.2nd
AND       F0009A
OR LOAD
AND LOAD
OUT       M02608	// OUT-BUFF R-UNLD-OK
OUTP      M02609	// OUT-BUFF R-UNLD-1P
; L52
LOAD      M02606	// OUT-BUFF L-UNLD-OK
OR        M02608	// OUT-BUFF R-UNLD-OK
OUT       M0260A	// UNLOAD-OK KP
// ========================   L   OUT BUFFER   ==========================
; L55
LOAD      M12080	// L_P&P CYCLE RUN
AND       M04200	// R_2nd_20 R Pos.1st
AND       P0002E	// L_OUT BUFF ROTA-P&P
AND NOT   P0009B	// L_OUT BUFFER DIE EJECTOR ON
AND       M04022	// L_P&P_02 Y Pos.3rd PLACE
AND       P00056	// L_P&P DOWN
AND       P00138	// L_P&P 5th EJECT ON
OR        M18322	// T)L_OUT BUFFER VC ON
OR        M18110	// L_OUT BUFFER VC ON
AND NOT   M18112	// L_OUT BUFFER VC OFF
AND NOT   M1812A	// AUAc¨ú©ªA¢¬©öC¡¤I BUFF VC OFF
AND NOT   M18324	// T)L_OUT BUFFER VC OFF
AND NOT   M19102	// T)LEFT INITIAL
OUT       M18110	// L_OUT BUFFER VC ON

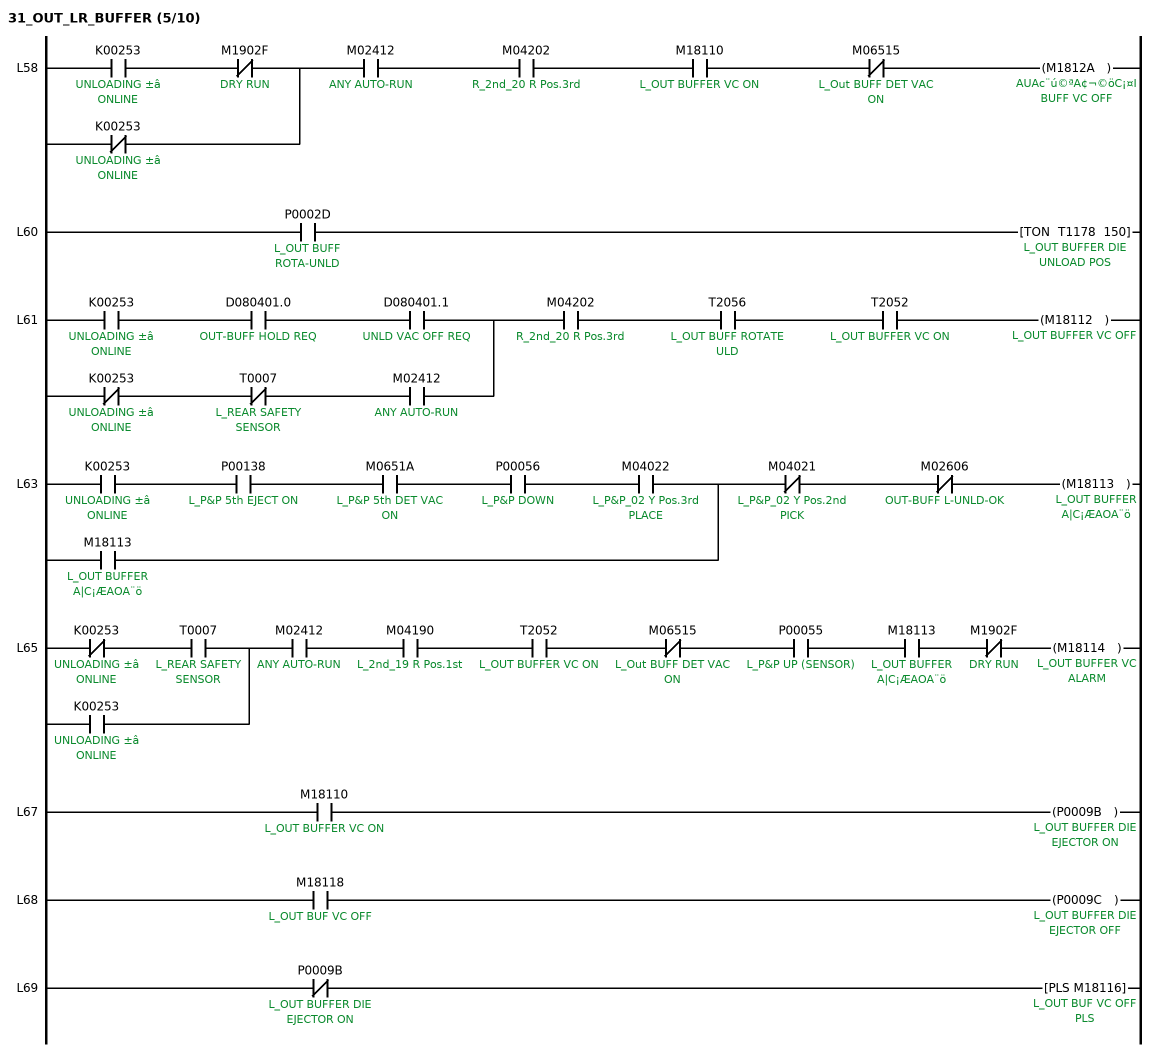
; L58
LOAD      K00253	// UNLOADING ±â ONLINE
AND NOT   M1902F	// DRY RUN
OR NOT    K00253	// UNLOADING ±â ONLINE
AND       M02412	// ANY AUTO-RUN
AND       M04202	// R_2nd_20 R Pos.3rd
AND       M18110	// L_OUT BUFFER VC ON
AND NOT   M06515	// L_Out BUFF DET VAC ON
OUT       M1812A	// AUAc¨ú©ªA¢¬©öC¡¤I BUFF VC OFF
; L60
LOAD      P0002D	// L_OUT BUFF ROTA-UNLD
TON       T1178 150	// L_OUT BUFFER DIE UNLOAD POS
; L61
LOAD      K00253	// UNLOADING ±â ONLINE
AND       D080401.0	// OUT-BUFF HOLD REQ
AND       D080401.1	// UNLD VAC OFF REQ
LOAD NOT  K00253	// UNLOADING ±â ONLINE
AND NOT   T0007	// L_REAR SAFETY SENSOR
AND       M02412	// ANY AUTO-RUN
OR LOAD
AND       M04202	// R_2nd_20 R Pos.3rd
AND       T2056	// L_OUT BUFF ROTATE     ULD
AND       T2052	// L_OUT BUFFER VC ON
OUT       M18112	// L_OUT BUFFER VC OFF
; L63
LOAD      K00253	// UNLOADING ±â ONLINE
AND       P00138	// L_P&P 5th EJECT ON
AND       M0651A	// L_P&P 5th DET VAC ON
AND       P00056	// L_P&P DOWN
AND       M04022	// L_P&P_02 Y Pos.3rd PLACE
OR        M18113	// L_OUT BUFFER A|C¡ÆAOA¨ö
AND NOT   M04021	// L_P&P_02 Y Pos.2nd PICK
AND NOT   M02606	// OUT-BUFF L-UNLD-OK
OUT       M18113	// L_OUT BUFFER A|C¡ÆAOA¨ö
; L65
LOAD NOT  K00253	// UNLOADING ±â ONLINE
AND       T0007	// L_REAR SAFETY SENSOR
OR        K00253	// UNLOADING ±â ONLINE
AND       M02412	// ANY AUTO-RUN
AND       M04190	// L_2nd_19 R Pos.1st 
AND       T2052	// L_OUT BUFFER VC ON
AND NOT   M06515	// L_Out BUFF DET VAC ON
AND       P00055	// L_P&P UP (SENSOR)
AND       M18113	// L_OUT BUFFER A|C¡ÆAOA¨ö
AND NOT   M1902F	// DRY RUN
OUT       M18114	// L_OUT BUFFER VC ALARM
; L67
LOAD      M18110	// L_OUT BUFFER VC ON
OUT       P0009B	// L_OUT BUFFER DIE EJECTOR ON
; L68
LOAD      M18118	// L_OUT BUF VC OFF
OUT       P0009C	// L_OUT BUFFER DIE EJECTOR OFF
; L69
LOAD NOT  P0009B	// L_OUT BUFFER DIE EJECTOR ON
OUTP      M18116	// L_OUT BUF VC OFF PLS

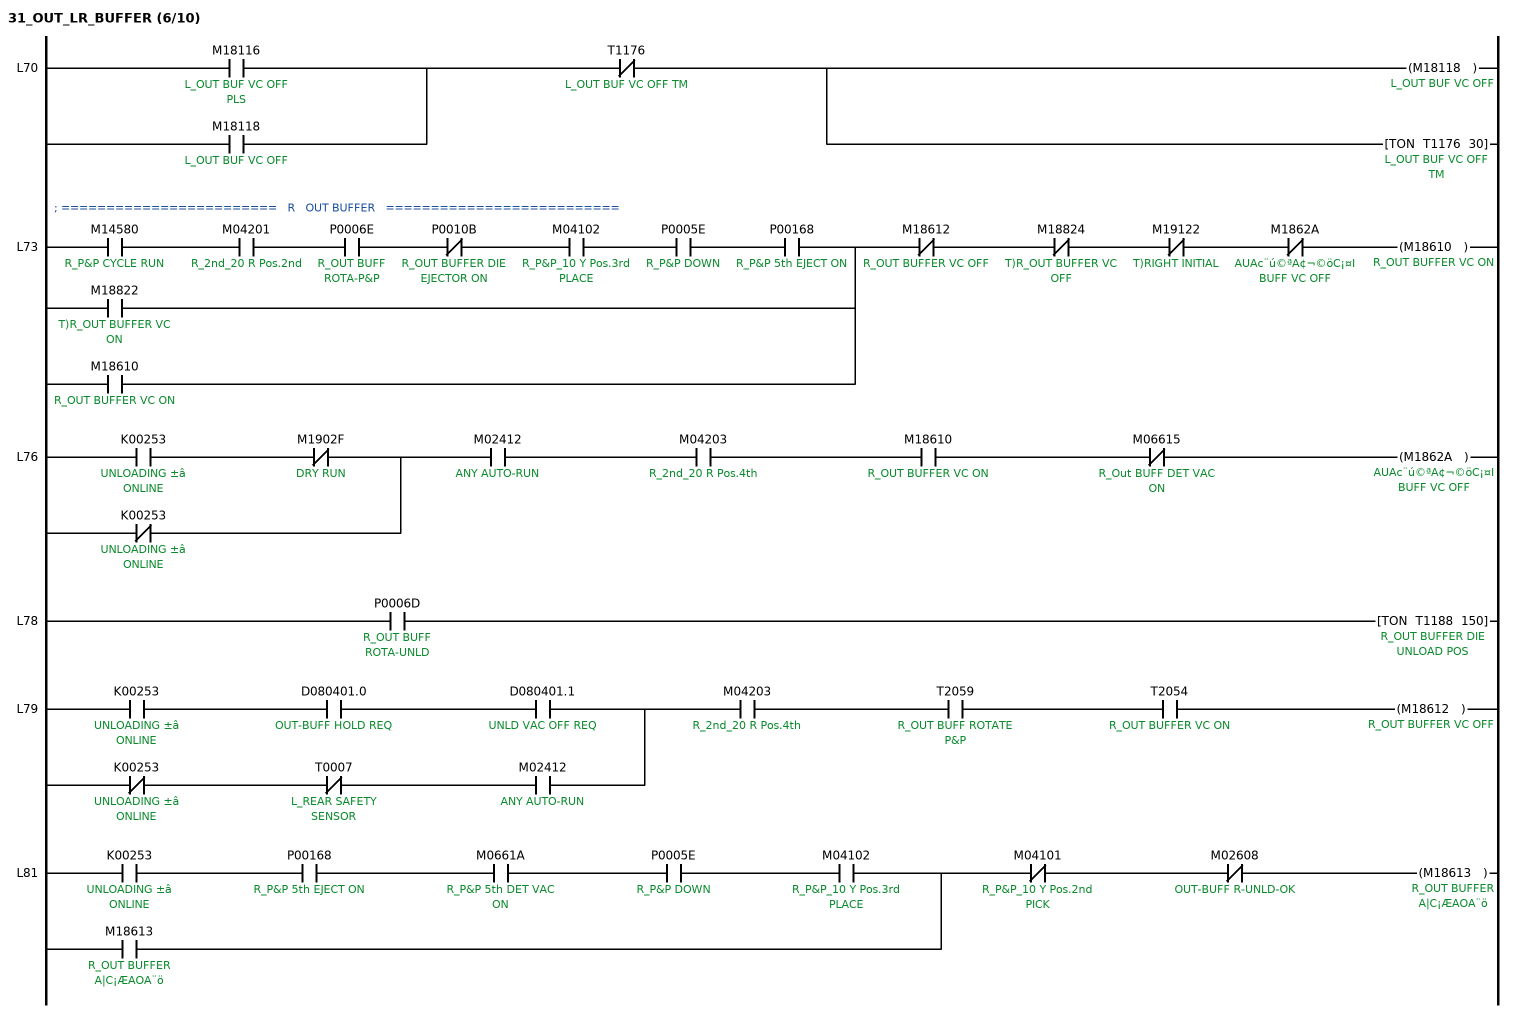
; L70
LOAD      M18116	// L_OUT BUF VC OFF PLS
OR        M18118	// L_OUT BUF VC OFF
AND NOT   T1176	// L_OUT BUF VC OFF TM
OUT       M18118	// L_OUT BUF VC OFF
TON       T1176 30	// L_OUT BUF VC OFF TM
// ========================   R   OUT BUFFER   ==========================
; L73
LOAD      M14580	// R_P&P CYCLE RUN
AND       M04201	// R_2nd_20 R Pos.2nd
AND       P0006E	// R_OUT BUFF ROTA-P&P
AND NOT   P0010B	// R_OUT BUFFER DIE EJECTOR ON
AND       M04102	// R_P&P_10 Y Pos.3rd PLACE
AND       P0005E	// R_P&P DOWN
AND       P00168	// R_P&P 5th EJECT ON
OR        M18822	// T)R_OUT BUFFER VC ON
OR        M18610	// R_OUT BUFFER VC ON
AND NOT   M18612	// R_OUT BUFFER VC OFF
AND NOT   M18824	// T)R_OUT BUFFER VC OFF
AND NOT   M19122	// T)RIGHT INITIAL
AND NOT   M1862A	// AUAc¨ú©ªA¢¬©öC¡¤I BUFF VC OFF
OUT       M18610	// R_OUT BUFFER VC ON
; L76
LOAD      K00253	// UNLOADING ±â ONLINE
AND NOT   M1902F	// DRY RUN
OR NOT    K00253	// UNLOADING ±â ONLINE
AND       M02412	// ANY AUTO-RUN
AND       M04203	// R_2nd_20 R Pos.4th 
AND       M18610	// R_OUT BUFFER VC ON
AND NOT   M06615	// R_Out BUFF DET VAC ON
OUT       M1862A	// AUAc¨ú©ªA¢¬©öC¡¤I BUFF VC OFF
; L78
LOAD      P0006D	// R_OUT BUFF ROTA-UNLD
TON       T1188 150	// R_OUT BUFFER DIE UNLOAD POS
; L79
LOAD      K00253	// UNLOADING ±â ONLINE
AND       D080401.0	// OUT-BUFF HOLD REQ
AND       D080401.1	// UNLD VAC OFF REQ
LOAD NOT  K00253	// UNLOADING ±â ONLINE
AND NOT   T0007	// L_REAR SAFETY SENSOR
AND       M02412	// ANY AUTO-RUN
OR LOAD
AND       M04203	// R_2nd_20 R Pos.4th 
AND       T2059	// R_OUT BUFF ROTATE      P&P
AND       T2054	// R_OUT BUFFER VC ON
OUT       M18612	// R_OUT BUFFER VC OFF
; L81
LOAD      K00253	// UNLOADING ±â ONLINE
AND       P00168	// R_P&P 5th EJECT ON
AND       M0661A	// R_P&P 5th DET VAC ON
AND       P0005E	// R_P&P DOWN
AND       M04102	// R_P&P_10 Y Pos.3rd PLACE
OR        M18613	// R_OUT BUFFER A|C¡ÆAOA¨ö
AND NOT   M04101	// R_P&P_10 Y Pos.2nd PICK
AND NOT   M02608	// OUT-BUFF R-UNLD-OK
OUT       M18613	// R_OUT BUFFER A|C¡ÆAOA¨ö

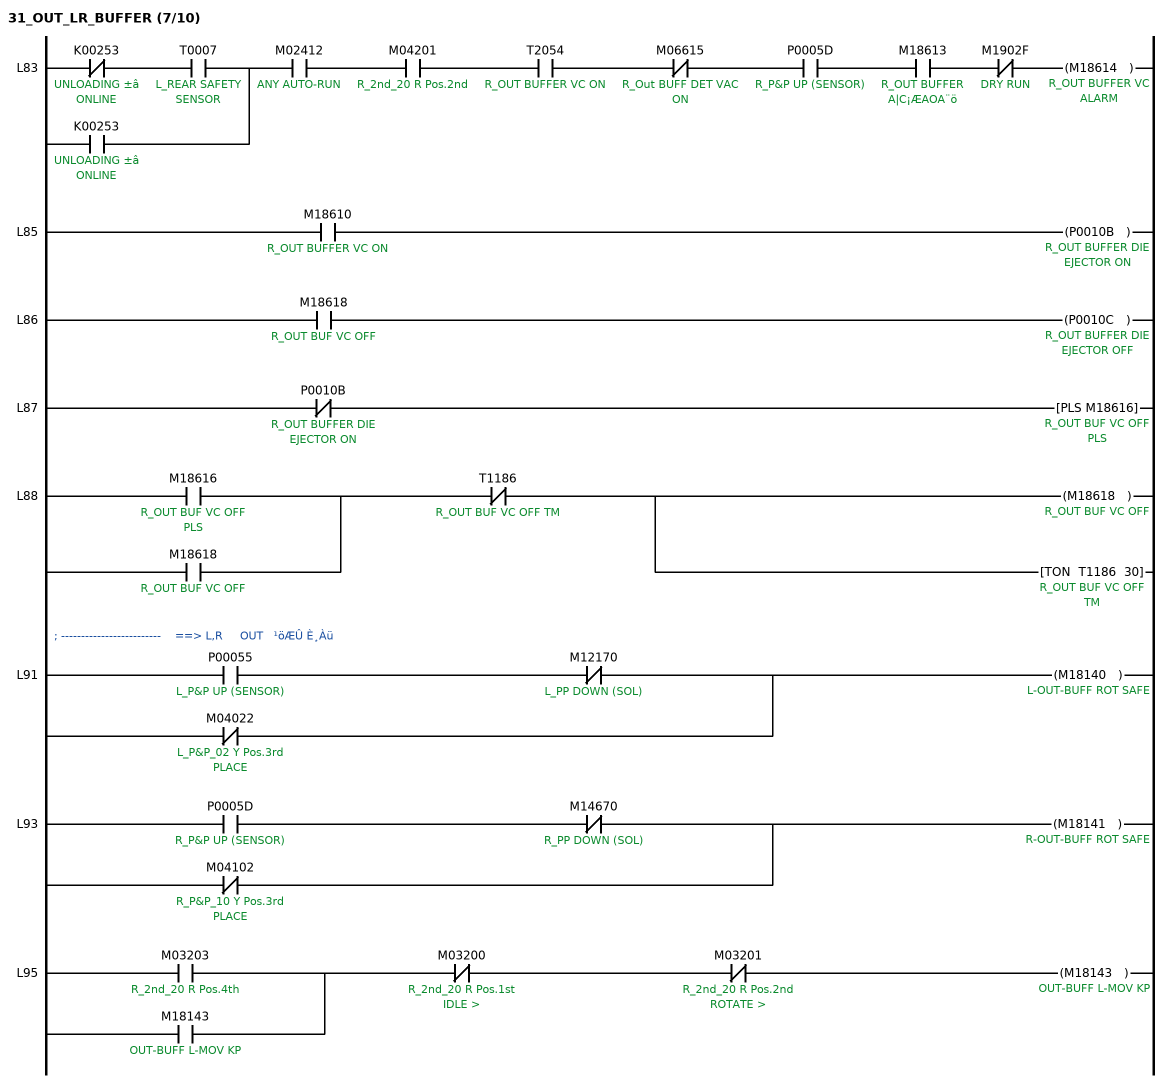
; L83
LOAD NOT  K00253	// UNLOADING ±â ONLINE
AND       T0007	// L_REAR SAFETY SENSOR
OR        K00253	// UNLOADING ±â ONLINE
AND       M02412	// ANY AUTO-RUN
AND       M04201	// R_2nd_20 R Pos.2nd
AND       T2054	// R_OUT BUFFER VC ON
AND NOT   M06615	// R_Out BUFF DET VAC ON
AND       P0005D	// R_P&P UP (SENSOR)
AND       M18613	// R_OUT BUFFER A|C¡ÆAOA¨ö
AND NOT   M1902F	// DRY RUN
OUT       M18614	// R_OUT BUFFER VC ALARM
; L85
LOAD      M18610	// R_OUT BUFFER VC ON
OUT       P0010B	// R_OUT BUFFER DIE EJECTOR ON
; L86
LOAD      M18618	// R_OUT BUF VC OFF
OUT       P0010C	// R_OUT BUFFER DIE EJECTOR OFF
; L87
LOAD NOT  P0010B	// R_OUT BUFFER DIE EJECTOR ON
OUTP      M18616	// R_OUT BUF VC OFF PLS
; L88
LOAD      M18616	// R_OUT BUF VC OFF PLS
OR        M18618	// R_OUT BUF VC OFF
AND NOT   T1186	// R_OUT BUF VC OFF TM
OUT       M18618	// R_OUT BUF VC OFF
TON       T1186 30	// R_OUT BUF VC OFF TM
// -------------------------    ==> L,R     OUT   ¹öÆÛ È¸Àü
; L91
LOAD      P00055	// L_P&P UP (SENSOR)
AND NOT   M12170	// L_PP DOWN (SOL)
OR NOT    M04022	// L_P&P_02 Y Pos.3rd PLACE
OUT       M18140	// L-OUT-BUFF ROT SAFE
; L93
LOAD      P0005D	// R_P&P UP (SENSOR)
AND NOT   M14670	// R_PP DOWN (SOL)
OR NOT    M04102	// R_P&P_10 Y Pos.3rd PLACE
OUT       M18141	// R-OUT-BUFF ROT SAFE
; L95
LOAD      M03203	// R_2nd_20 R Pos.4th 
OR        M18143	// OUT-BUFF L-MOV KP
AND NOT   M03200	// R_2nd_20 R Pos.1st IDLE >
AND NOT   M03201	// R_2nd_20 R Pos.2nd ROTATE >
OUT       M18143	// OUT-BUFF L-MOV KP

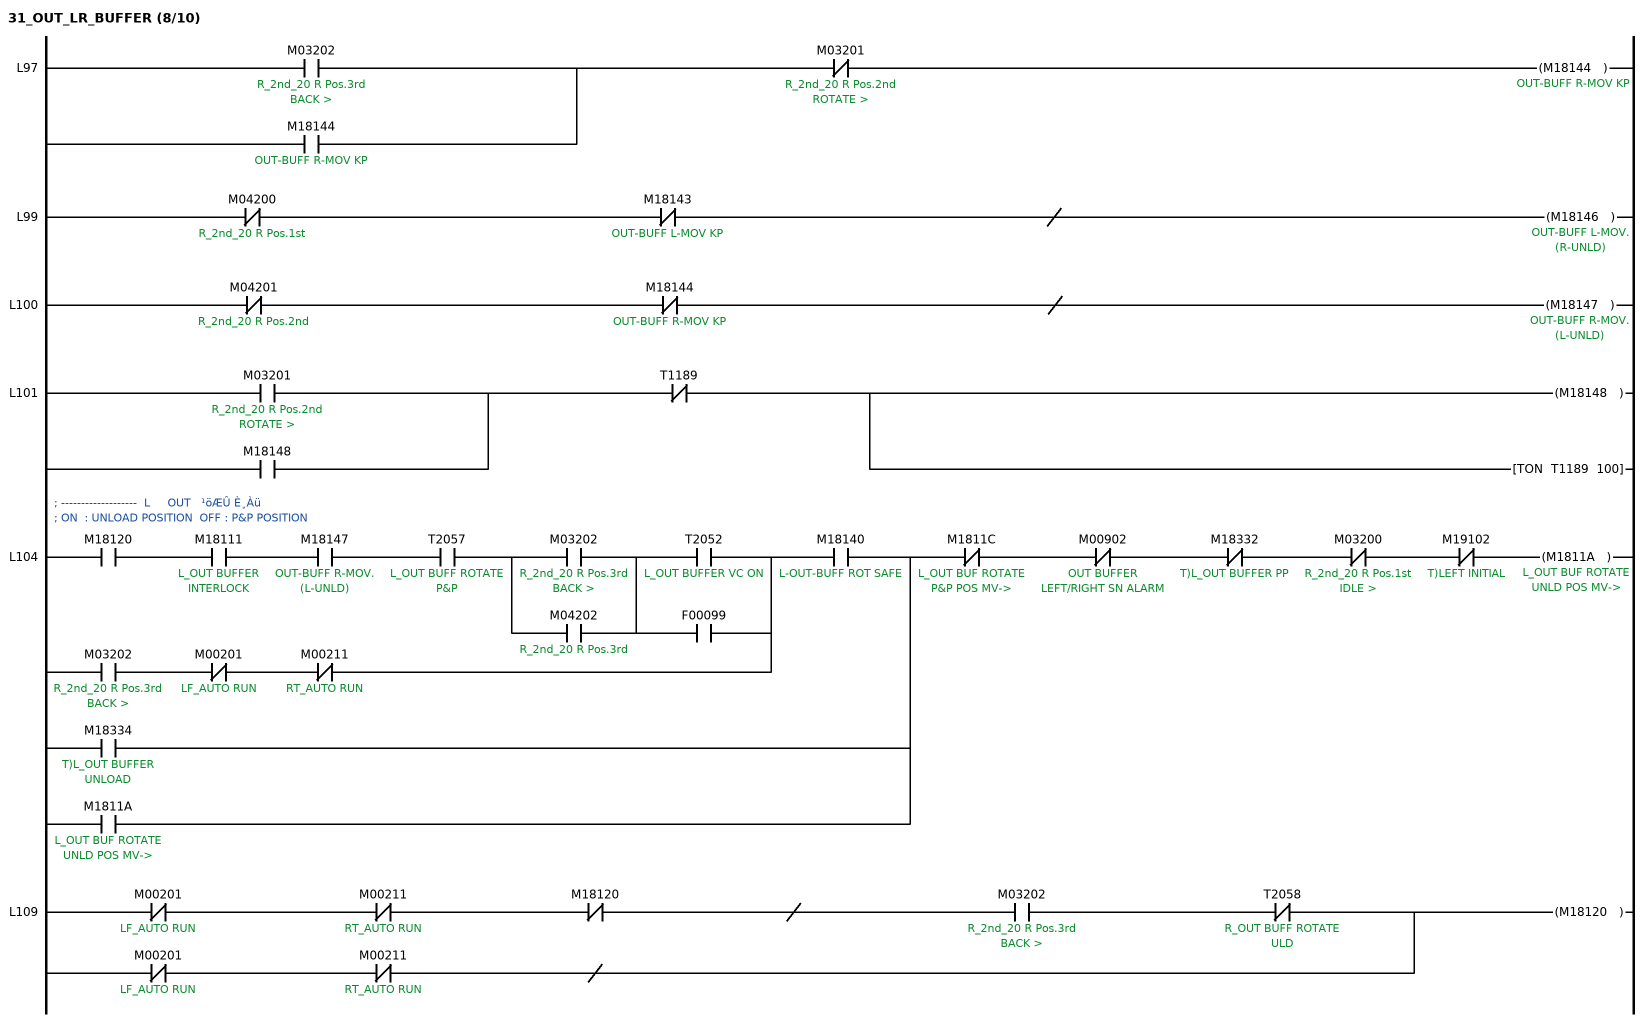
; L97
LOAD      M03202	// R_2nd_20 R Pos.3rd BACK >
OR        M18144	// OUT-BUFF R-MOV KP
AND NOT   M03201	// R_2nd_20 R Pos.2nd ROTATE >
OUT       M18144	// OUT-BUFF R-MOV KP
; L99
LOAD NOT  M04200	// R_2nd_20 R Pos.1st
AND NOT   M18143	// OUT-BUFF L-MOV KP
NOT
OUT       M18146	// OUT-BUFF L-MOV.  (R-UNLD)
; L100
LOAD NOT  M04201	// R_2nd_20 R Pos.2nd
AND NOT   M18144	// OUT-BUFF R-MOV KP
NOT
OUT       M18147	// OUT-BUFF R-MOV.  (L-UNLD)
; L101
LOAD      M03201	// R_2nd_20 R Pos.2nd ROTATE >
OR        M18148
AND NOT   T1189
OUT       M18148
TON       T1189 100
// -------------------  L     OUT   ¹öÆÛ È¸Àü
; L104
LOAD      M18120
AND       M18111	// L_OUT BUFFER INTERLOCK
AND       M18147	// OUT-BUFF R-MOV.  (L-UNLD)
AND       T2057	// L_OUT BUFF ROTATE      P&P
LOAD      M03202	// R_2nd_20 R Pos.3rd BACK >
OR        M04202	// R_2nd_20 R Pos.3rd
AND LOAD
LOAD      T2052	// L_OUT BUFFER VC ON
OR        F00099
AND LOAD
LOAD      M03202	// R_2nd_20 R Pos.3rd BACK >
AND NOT   M00201	// LF_AUTO RUN
AND NOT   M00211	// RT_AUTO RUN
OR LOAD
AND       M18140	// L-OUT-BUFF ROT SAFE
OR        M18334	// T)L_OUT BUFFER UNLOAD
OR        M1811A	// L_OUT BUF ROTATE UNLD POS MV->
AND NOT   M1811C	// L_OUT BUF ROTATE P&P POS MV->
AND NOT   M00902	// OUT BUFFER LEFT/RIGHT SN ALARM
AND NOT   M18332	// T)L_OUT BUFFER PP
AND NOT   M03200	// R_2nd_20 R Pos.1st IDLE >
AND NOT   M19102	// T)LEFT INITIAL
OUT       M1811A	// L_OUT BUF ROTATE UNLD POS MV->
// output comment: ON  : UNLOAD POSITION  OFF : P&P POSITION
; L109
LOAD NOT  M00201	// LF_AUTO RUN
AND NOT   M00211	// RT_AUTO RUN
AND NOT   M18120
NOT
AND       M03202	// R_2nd_20 R Pos.3rd BACK >
AND NOT   T2058	// R_OUT BUFF ROTATE      ULD
LOAD NOT  M00201	// LF_AUTO RUN
AND NOT   M00211	// RT_AUTO RUN
NOT
OR LOAD
OUT       M18120

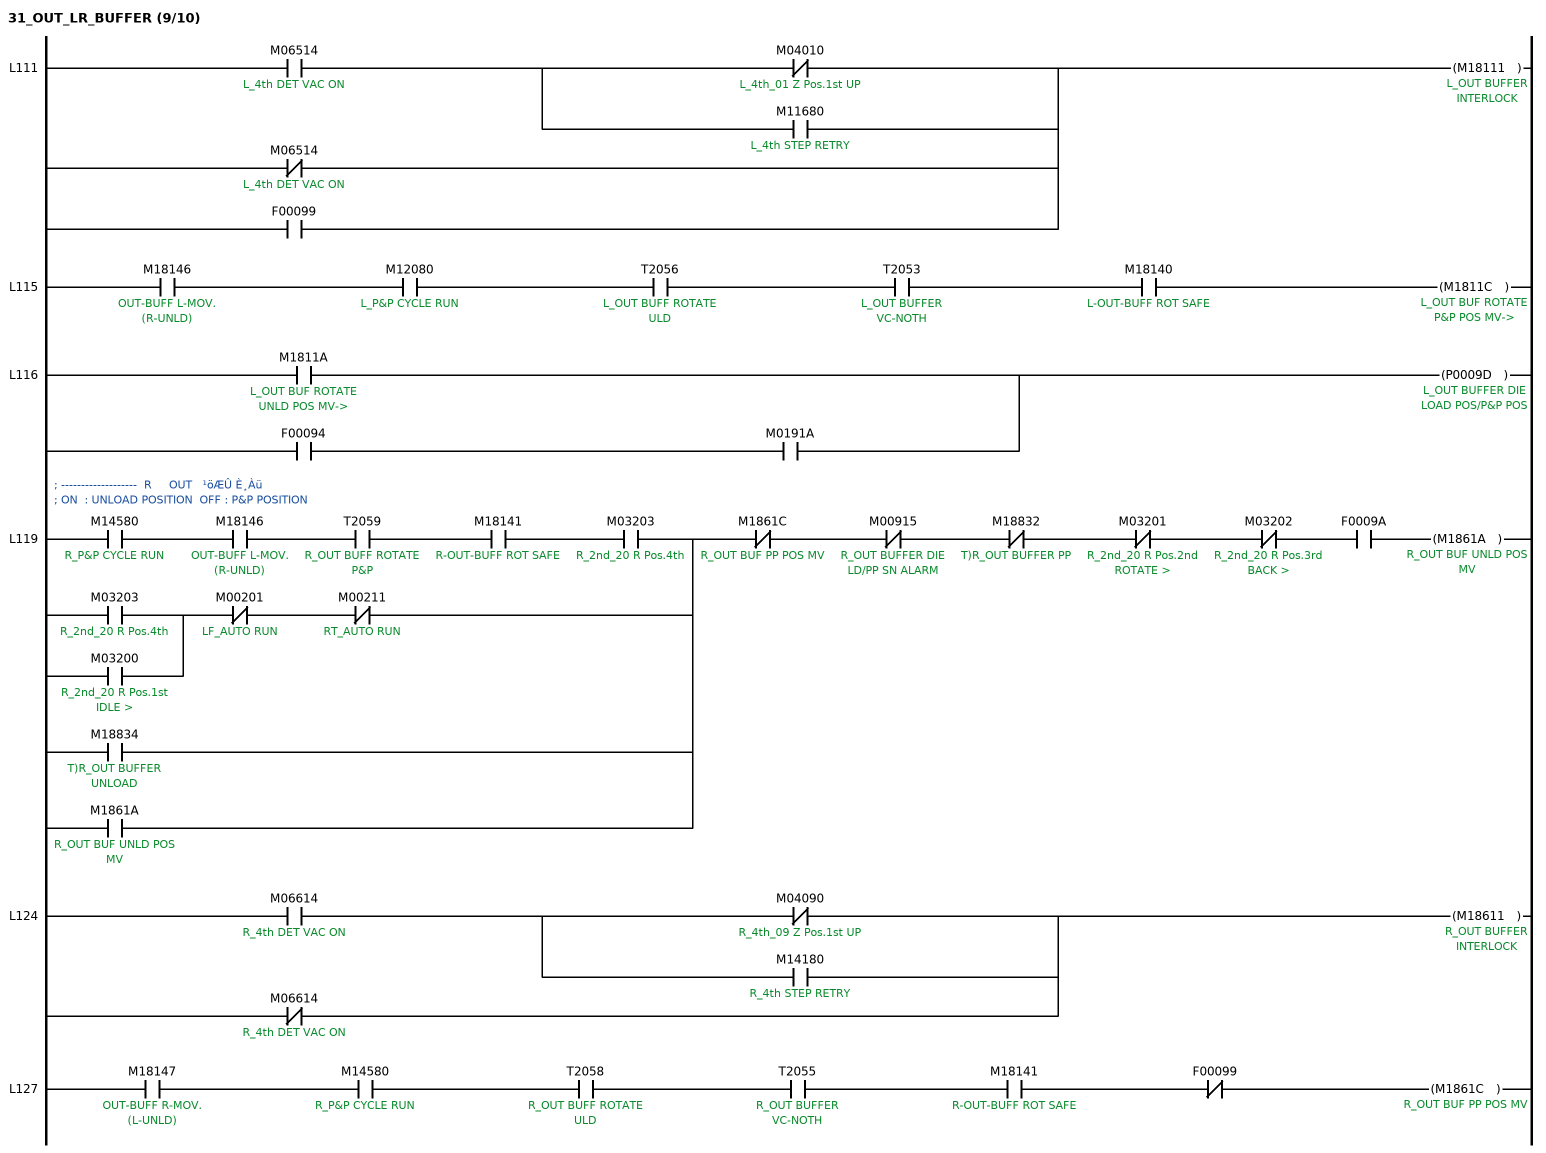
; L111
LOAD      M06514	// L_4th DET VAC ON
LOAD NOT  M04010	// L_4th_01 Z Pos.1st UP
OR        M11680	// L_4th STEP RETRY
AND LOAD
OR NOT    M06514	// L_4th DET VAC ON
OR        F00099
OUT       M18111	// L_OUT BUFFER INTERLOCK
; L115
LOAD      M18146	// OUT-BUFF L-MOV.  (R-UNLD)
AND       M12080	// L_P&P CYCLE RUN
AND       T2056	// L_OUT BUFF ROTATE     ULD
AND       T2053	// L_OUT BUFFER VC-NOTH
AND       M18140	// L-OUT-BUFF ROT SAFE
OUT       M1811C	// L_OUT BUF ROTATE P&P POS MV->
; L116
LOAD      M1811A	// L_OUT BUF ROTATE UNLD POS MV->
LOAD      F00094
AND       M0191A
OR LOAD
OUT       P0009D	// L_OUT BUFFER DIE LOAD POS/P&P POS
// -------------------  R     OUT   ¹öÆÛ È¸Àü
; L119
LOAD      M14580	// R_P&P CYCLE RUN
AND       M18146	// OUT-BUFF L-MOV.  (R-UNLD)
AND       T2059	// R_OUT BUFF ROTATE      P&P
AND       M18141	// R-OUT-BUFF ROT SAFE
AND       M03203	// R_2nd_20 R Pos.4th 
LOAD      M03203	// R_2nd_20 R Pos.4th 
OR        M03200	// R_2nd_20 R Pos.1st IDLE >
AND NOT   M00201	// LF_AUTO RUN
AND NOT   M00211	// RT_AUTO RUN
OR LOAD
OR        M18834	// T)R_OUT BUFFER UNLOAD
OR        M1861A	// R_OUT BUF UNLD POS MV
AND NOT   M1861C	// R_OUT BUF PP POS MV
AND NOT   M00915	// R_OUT BUFFER DIE LD/PP SN ALARM
AND NOT   M18832	// T)R_OUT BUFFER PP
AND NOT   M03201	// R_2nd_20 R Pos.2nd ROTATE >
AND NOT   M03202	// R_2nd_20 R Pos.3rd BACK >
AND       F0009A
OUT       M1861A	// R_OUT BUF UNLD POS MV
// output comment: ON  : UNLOAD POSITION  OFF : P&P POSITION
; L124
LOAD      M06614	// R_4th DET VAC ON
LOAD NOT  M04090	// R_4th_09 Z Pos.1st UP
OR        M14180	// R_4th STEP RETRY
AND LOAD
OR NOT    M06614	// R_4th DET VAC ON
OUT       M18611	// R_OUT BUFFER INTERLOCK
; L127
LOAD      M18147	// OUT-BUFF R-MOV.  (L-UNLD)
AND       M14580	// R_P&P CYCLE RUN
AND       T2058	// R_OUT BUFF ROTATE      ULD
AND       T2055	// R_OUT BUFFER VC-NOTH
AND       M18141	// R-OUT-BUFF ROT SAFE
AND NOT   F00099
OUT       M1861C	// R_OUT BUF PP POS MV

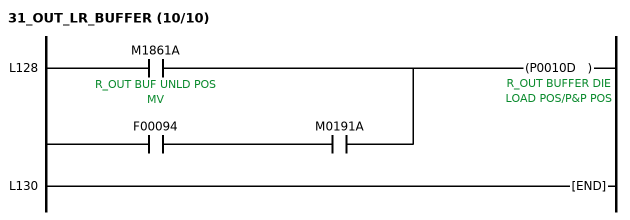
; L128
LOAD      M1861A	// R_OUT BUF UNLD POS MV
LOAD      F00094
AND       M0191A
OR LOAD
OUT       P0010D	// R_OUT BUFFER DIE LOAD POS/P&P POS
; L130
END

PROGRAM 40_2D_CODE (task: ½ºÄµ ÇÁ·Î±×·¥)

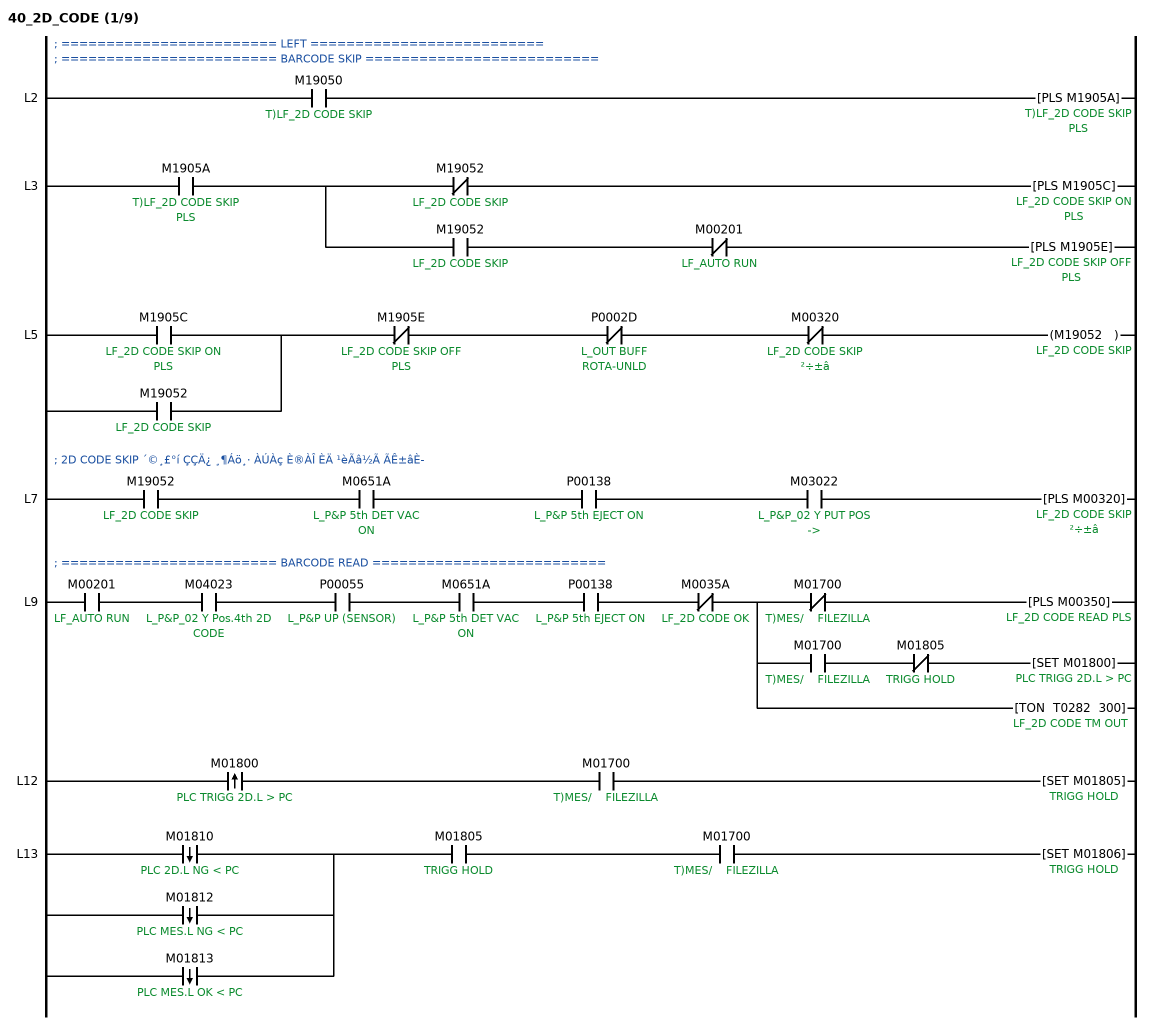
// ======================== LEFT ==========================
// ======================== BARCODE SKIP ==========================
; L2
LOAD      M19050	// T)LF_2D CODE SKIP
OUTP      M1905A	// T)LF_2D CODE SKIP PLS
; L3
LOAD      M1905A	// T)LF_2D CODE SKIP PLS
MPUSH
AND NOT   M19052	// LF_2D CODE SKIP
OUTP      M1905C	// LF_2D CODE SKIP ON PLS
MPOP
AND       M19052	// LF_2D CODE SKIP
AND NOT   M00201	// LF_AUTO RUN
OUTP      M1905E	// LF_2D CODE SKIP OFF PLS
; L5
LOAD      M1905C	// LF_2D CODE SKIP ON PLS
OR        M19052	// LF_2D CODE SKIP
AND NOT   M1905E	// LF_2D CODE SKIP OFF PLS
AND NOT   P0002D	// L_OUT BUFF ROTA-UNLD
AND NOT   M00320	// LF_2D CODE SKIP ²÷±â
OUT       M19052	// LF_2D CODE SKIP
; L7
LOAD      M19052	// LF_2D CODE SKIP
AND       M0651A	// L_P&P 5th DET VAC ON
AND       P00138	// L_P&P 5th EJECT ON
AND       M03022	// L_P&P_02 Y PUT POS ->
OUTP      M00320	// LF_2D CODE SKIP ²÷±â
// output comment: 2D CODE SKIP ´©¸£°í ÇÇÄ¿ ¸¶Áö¸· ÀÚÀç È®ÀÎ ÈÄ ¹èÃâ½Ã ÃÊ±âÈ­
// ======================== BARCODE READ ==========================
; L9
LOAD      M00201	// LF_AUTO RUN
AND       M04023	// L_P&P_02 Y Pos.4th 2D CODE
AND       P00055	// L_P&P UP (SENSOR)
AND       M0651A	// L_P&P 5th DET VAC ON
AND       P00138	// L_P&P 5th EJECT ON
AND NOT   M0035A	// LF_2D CODE OK
MPUSH
AND NOT   M01700	// T)MES/    FILEZILLA
OUTP      M00350	// LF_2D CODE READ PLS
MLOAD
AND       M01700	// T)MES/    FILEZILLA
AND NOT   M01805	// TRIGG HOLD
SET       M01800	// PLC TRIGG 2D.L > PC
MPOP
TON       T0282 300	// LF_2D CODE TM OUT
; L12
LOADP     M01800	// PLC TRIGG 2D.L > PC
AND       M01700	// T)MES/    FILEZILLA
SET       M01805	// TRIGG HOLD
; L13
LOADN     M01810	// PLC 2D.L NG < PC
ORN       M01812	// PLC MES.L NG < PC
ORN       M01813	// PLC MES.L OK < PC
AND       M01805	// TRIGG HOLD
AND       M01700	// T)MES/    FILEZILLA
SET       M01806	// TRIGG HOLD

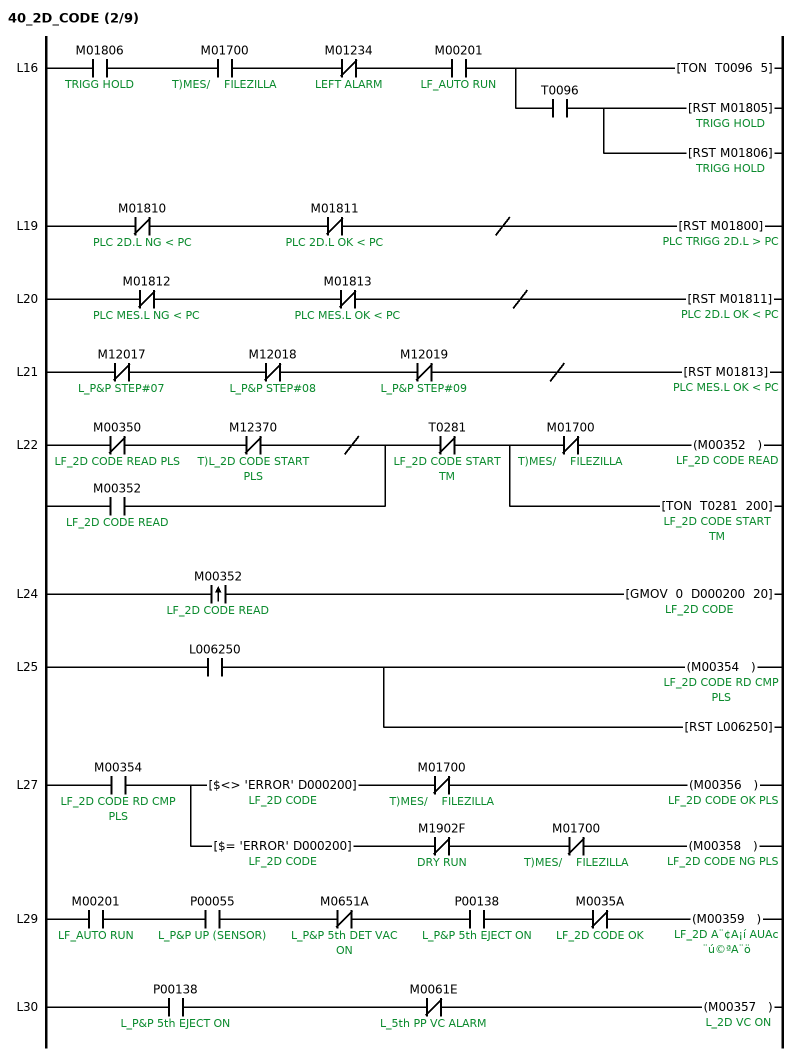
; L16
LOAD      M01806	// TRIGG HOLD
AND       M01700	// T)MES/    FILEZILLA
AND NOT   M01234	// LEFT ALARM
AND       M00201	// LF_AUTO RUN
TON       T0096 5
AND       T0096
RST       M01805	// TRIGG HOLD
RST       M01806	// TRIGG HOLD
; L19
LOAD NOT  M01810	// PLC 2D.L NG < PC
AND NOT   M01811	// PLC 2D.L OK < PC
NOT
RST       M01800	// PLC TRIGG 2D.L > PC
; L20
LOAD NOT  M01812	// PLC MES.L NG < PC
AND NOT   M01813	// PLC MES.L OK < PC
NOT
RST       M01811	// PLC 2D.L OK < PC
; L21
LOAD NOT  M12017	// L_P&P STEP#07
AND NOT   M12018	// L_P&P STEP#08
AND NOT   M12019	// L_P&P STEP#09
NOT
RST       M01813	// PLC MES.L OK < PC
; L22
LOAD NOT  M00350	// LF_2D CODE READ PLS
AND NOT   M12370	// T)L_2D CODE START PLS
NOT
OR        M00352	// LF_2D CODE READ
AND NOT   T0281	// LF_2D CODE START TM
MPUSH
AND NOT   M01700	// T)MES/    FILEZILLA
OUT       M00352	// LF_2D CODE READ
MPOP
TON       T0281 200	// LF_2D CODE START TM
; L24
LOADP     M00352	// LF_2D CODE READ
GMOV      0 D000200 20	// LF_2D CODE
; L25
LOAD      L006250
OUT       M00354	// LF_2D CODE RD CMP PLS
RST       L006250
; L27
LOAD      M00354	// LF_2D CODE RD CMP PLS
MPUSH
AND$<>    'ERROR' D000200	// LF_2D CODE
AND NOT   M01700	// T)MES/    FILEZILLA
OUT       M00356	// LF_2D CODE OK PLS
MPOP
AND$=     'ERROR' D000200	// LF_2D CODE
AND NOT   M1902F	// DRY RUN
AND NOT   M01700	// T)MES/    FILEZILLA
OUT       M00358	// LF_2D CODE NG PLS
; L29
LOAD      M00201	// LF_AUTO RUN
AND       P00055	// L_P&P UP (SENSOR)
AND NOT   M0651A	// L_P&P 5th DET VAC ON
AND       P00138	// L_P&P 5th EJECT ON
AND NOT   M0035A	// LF_2D CODE OK
OUT       M00359	// LF_2D A¨¢A¡í AUAc ¨ú©ªA¨ö
; L30
LOAD      P00138	// L_P&P 5th EJECT ON
AND NOT   M0061E	// L_5th PP VC ALARM
OUT       M00357	// L_2D VC ON

